   1:  PR[91,1] = PR[90,1] + -92.039;
   1:  PR[91,2] = PR[90,2] + -4.496;
   1:L PR[91] R[100]mm/sec CNT100;
   1:  PR[91,1] = PR[90,1] + -90.857;
   1:  PR[91,2] = PR[90,2] + -8.105;
   1:L PR[91] R[100]mm/sec CNT100;
   1:  PR[91,1] = PR[90,1] + -88.939;
   1:  PR[91,2] = PR[90,2] + -11.398;
   1:L PR[91] R[100]mm/sec CNT100TB   .50sec,CALL END_PUD;
   1:  PR[92] = PR[91];
   1:  PR[92,3] = PR[92,3] + 20;
   1:J PR[92] 10% FINE;
   1:  PR[91] = PR[90];
   1:  PR[91,1] = PR[90,1] + 75.472;
   1:  PR[91,2] = PR[90,2] + -19.127;
   1:  PR[91,3] = PR[90,3] + 22.295;
   1:  PR[92] = PR[91];
   1:  PR[92,3] = PR[92,3] + 20;
   1:J PR[92] 10% FINE;
   1:L PR[91] R[100]mm/sec CNT100;
   1:  CALL LASER_DRAHT_START;
   1:  PR[91,1] = PR[90,1] + 77.707;
   1:  PR[91,2] = PR[90,2] + -18.824;
   1:L PR[91] R[100]mm/sec CNT100;
   1:  PR[91,1] = PR[90,1] + 79.977;
   1:  PR[91,2] = PR[90,2] + -18.016;
   1:L PR[91] R[100]mm/sec CNT100;
   1:  PR[91,1] = PR[90,1] + 81.671;
   1:  PR[91,2] = PR[90,2] + -17.392;
   1:L PR[91] R[100]mm/sec CNT100;
   1:  PR[91,1] = PR[90,1] + 83.993;
   1:  PR[91,2] = PR[90,2] + -15.925;
   1:L PR[91] R[100]mm/sec CNT100;
   1:  PR[91,1] = PR[90,1] + 85.202;
   1:  PR[91,2] = PR[90,2] + -15.146;
   1:L PR[91] R[100]mm/sec CNT100;
   1:  PR[91,1] = PR[90,1] + 88.142;
   1:  PR[91,2] = PR[90,2] + -12.194;
   1:L PR[91] R[100]mm/sec CNT100;
   1:  PR[91,1] = PR[90,1] + 90.342;
   1:  PR[91,2] = PR[90,2] + -8.694;
   1:L PR[91] R[100]mm/sec CNT100;
   1:  PR[91,1] = PR[90,1] + 91.704;
   1:  PR[91,2] = PR[90,2] + -4.807;
   1:L PR[91] R[100]mm/sec CNT100;
   1:  PR[91,1] = PR[90,1] + 92.097;
   1:  PR[91,2] = PR[90,2] + -1.400;
   1:L PR[91] R[100]mm/sec CNT100;
   1:  PR[91,1] = PR[90,1] + 92.205;
   1:  PR[91,2] = PR[90,2] + -0.692;
   1:L PR[91] R[100]mm/sec CNT100;
   1:  PR[91,1] = PR[90,1] + 91.906;
   1:  PR[91,2] = PR[90,2] + 1.920;
   1:L PR[91] R[100]mm/sec CNT100;
   1:  PR[91,1] = PR[90,1] + 91.796;
   1:  PR[91,2] = PR[90,2] + 2.516;
   1:L PR[91] R[100]mm/sec CNT100;
   1:  PR[91,1] = PR[90,1] + 91.703;
   1:  PR[91,2] = PR[90,2] + 3.353;
   1:L PR[91] R[100]mm/sec CNT100;
   1:  PR[91,1] = PR[90,1] + 90.342;
   1:  PR[91,2] = PR[90,2] + 7.235;
   1:L PR[91] R[100]mm/sec CNT100;
   1:  PR[91,1] = PR[90,1] + 88.142;
   1:  PR[91,2] = PR[90,2] + 10.735;
   1:L PR[91] R[100]mm/sec CNT100;
   1:  PR[91,1] = PR[90,1] + 85.209;
   1:  PR[91,2] = PR[90,2] + 13.680;
   1:L PR[91] R[100]mm/sec CNT100;
   1:  PR[91,1] = PR[90,1] + 82.872;
   1:  PR[91,2] = PR[90,2] + 15.154;
   1:L PR[91] R[100]mm/sec CNT100;
   1:  PR[91,1] = PR[90,1] + 81.671;
   1:  PR[91,2] = PR[90,2] + 15.930;
   1:L PR[91] R[100]mm/sec CNT100;
   1:  PR[91,1] = PR[90,1] + 79.341;
   1:  PR[91,2] = PR[90,2] + 16.758;
   1:L PR[91] R[100]mm/sec CNT100;
   1:  PR[91,1] = PR[90,1] + 77.707;
   1:  PR[91,2] = PR[90,2] + 17.362;
   1:L PR[91] R[100]mm/sec CNT100;
   1:  PR[91,1] = PR[90,1] + 75.594;
   1:  PR[91,2] = PR[90,2] + 17.620;
   1:L PR[91] R[100]mm/sec CNT100;
   1:  PR[91,1] = PR[90,1] + 73.504;
   1:  PR[91,2] = PR[90,2] + 17.907;
   1:L PR[91] R[100]mm/sec CNT100;
   1:  PR[91,1] = PR[90,1] + 71.787;
   1:  PR[91,2] = PR[90,2] + 17.735;
   1:L PR[91] R[100]mm/sec CNT100;
   1:  PR[91,1] = PR[90,1] + 69.263;
   1:  PR[91,2] = PR[90,2] + 17.523;
   1:L PR[91] R[100]mm/sec CNT100;
   1:  PR[91,1] = PR[90,1] + 68.056;
   1:  PR[91,2] = PR[90,2] + 17.123;
   1:L PR[91] R[100]mm/sec CNT100;
   1:  PR[91,1] = PR[90,1] + 65.192;
   1:  PR[91,2] = PR[90,2] + 16.224;
   1:L PR[91] R[100]mm/sec CNT100;
   1:  PR[91,1] = PR[90,1] + 64.524;
   1:  PR[91,2] = PR[90,2] + 15.821;
   1:L PR[91] R[100]mm/sec CNT100;
   1:  PR[91,1] = PR[90,1] + 61.487;
   1:  PR[91,2] = PR[90,2] + 14.050;
   1:L PR[91] R[100]mm/sec CNT100;
   1:  PR[91,1] = PR[90,1] + 58.354;
   1:  PR[91,2] = PR[90,2] + 11.097;
   1:L PR[91] R[100]mm/sec CNT100;
   1:  PR[91,1] = PR[90,1] + 55.873;
   1:  PR[91,2] = PR[90,2] + 7.525;
   1:L PR[91] R[100]mm/sec CNT100;
   1:  PR[91,1] = PR[90,1] + 54.321;
   1:  PR[91,2] = PR[90,2] + 3.514;
   1:L PR[91] R[100]mm/sec CNT100;
   1:  PR[91,1] = PR[90,1] + 53.882;
   1:  PR[91,2] = PR[90,2] + 0.062;
   1:L PR[91] R[100]mm/sec CNT100;
   1:  PR[91,1] = PR[90,1] + 53.837;
   1:  PR[91,2] = PR[90,2] + -0.667;
   1:L PR[91] R[100]mm/sec CNT100;
   1:  PR[91,1] = PR[90,1] + 54.190;
   1:  PR[91,2] = PR[90,2] + -3.510;
   1:L PR[91] R[100]mm/sec CNT100;
   1:  PR[91,1] = PR[90,1] + 54.254;
   1:  PR[91,2] = PR[90,2] + -4.426;
   1:L PR[91] R[100]mm/sec CNT100;
   1:  PR[91,1] = PR[90,1] + 54.322;
   1:  PR[91,2] = PR[90,2] + -4.976;
   1:L PR[91] R[100]mm/sec CNT100;
   1:  PR[91,1] = PR[90,1] + 55.872;
   1:  PR[91,2] = PR[90,2] + -8.982;
   1:L PR[91] R[100]mm/sec CNT100;
   1:  PR[91,1] = PR[90,1] + 58.317;
   1:  PR[91,2] = PR[90,2] + -12.492;
   1:L PR[91] R[100]mm/sec CNT100;
   1:  PR[91,1] = PR[90,1] + 58.369;
   1:  PR[91,2] = PR[90,2] + -12.571;
   1:L PR[91] R[100]mm/sec CNT100;
   1:  PR[91,1] = PR[90,1] + 61.489;
   1:  PR[91,2] = PR[90,2] + -15.511;
   1:L PR[91] R[100]mm/sec CNT100;
   1:  PR[91,1] = PR[90,1] + 65.193;
   1:  PR[91,2] = PR[90,2] + -17.687;
   1:L PR[91] R[100]mm/sec CNT100;
   1:  PR[91,1] = PR[90,1] + 66.066;
   1:  PR[91,2] = PR[90,2] + -17.975;
   1:L PR[91] R[100]mm/sec CNT100;
   1:  PR[91,1] = PR[90,1] + 69.262;
   1:  PR[91,2] = PR[90,2] + -18.985;
   1:L PR[91] R[100]mm/sec CNT100;
   1:  PR[91,1] = PR[90,1] + 70.738;
   1:  PR[91,2] = PR[90,2] + -19.131;
   1:L PR[91] R[100]mm/sec CNT100;
   1:  PR[91,1] = PR[90,1] + 73.504;
   1:  PR[91,2] = PR[90,2] + -19.369;
   1:L PR[91] R[100]mm/sec CNT100;
   1:  PR[91,1] = PR[90,1] + 75.472;
   1:  PR[91,2] = PR[90,2] + -19.127;
   1:L PR[91] R[100]mm/sec CNT100TB   .50sec,CALL END_PUD;
   1:  PR[92] = PR[91];
   1:  PR[92,3] = PR[92,3] + 20;
   1:J PR[92] 10% FINE;
   1:  PR[91,1] = PR[90,1] + 37.828;
   1:  PR[91,2] = PR[90,2] + -13.861;
   1:  PR[92] = PR[91];
   1:  PR[92,3] = PR[92,3] + 20;
   1:J PR[92] 10% FINE;
   1:L PR[91] R[100]mm/sec CNT100;
   1:  CALL LASER_DRAHT_START;
   1:  PR[91,1] = PR[90,1] + 37.858;
   1:  PR[91,2] = PR[90,2] + -13.831;
   1:L PR[91] R[100]mm/sec CNT100;
   1:  PR[91,1] = PR[90,1] + 40.722;
   1:  PR[91,2] = PR[90,2] + -10.089;
   1:L PR[91] R[100]mm/sec CNT100;
   1:  PR[91,1] = PR[90,1] + 40.785;
   1:  PR[91,2] = PR[90,2] + -9.999;
   1:L PR[91] R[100]mm/sec CNT100;
   1:  PR[91,1] = PR[90,1] + 40.830;
   1:  PR[91,2] = PR[90,2] + -9.903;
   1:L PR[91] R[100]mm/sec CNT100;
   1:  PR[91,1] = PR[90,1] + 42.623;
   1:  PR[91,2] = PR[90,2] + -5.565;
   1:L PR[91] R[100]mm/sec CNT100;
   1:  PR[91,1] = PR[90,1] + 42.638;
   1:  PR[91,2] = PR[90,2] + -5.509;
   1:L PR[91] R[100]mm/sec CNT100;
   1:  PR[91,1] = PR[90,1] + 42.845;
   1:  PR[91,2] = PR[90,2] + -3.661;
   1:L PR[91] R[100]mm/sec CNT100;
   1:  PR[91,1] = PR[90,1] + 43.245;
   1:  PR[91,2] = PR[90,2] + -0.613;
   1:L PR[91] R[100]mm/sec CNT100;
   1:  PR[91,1] = PR[90,1] + 43.244;
   1:  PR[91,2] = PR[90,2] + -0.541;
   1:L PR[91] R[100]mm/sec CNT100;
   1:  PR[91,1] = PR[90,1] + 42.643;
   1:  PR[91,2] = PR[90,2] + 4.031;
   1:L PR[91] R[100]mm/sec CNT100;
   1:  PR[91,1] = PR[90,1] + 42.623;
   1:  PR[91,2] = PR[90,2] + 4.106;
   1:L PR[91] R[100]mm/sec CNT100;
   1:  PR[91,1] = PR[90,1] + 40.830;
   1:  PR[91,2] = PR[90,2] + 8.444;
   1:L PR[91] R[100]mm/sec CNT100;
   1:  PR[91,1] = PR[90,1] + 40.785;
   1:  PR[91,2] = PR[90,2] + 8.540;
   1:L PR[91] R[100]mm/sec CNT100;
   1:  PR[91,1] = PR[90,1] + 40.722;
   1:  PR[91,2] = PR[90,2] + 8.630;
   1:L PR[91] R[100]mm/sec CNT100;
   1:  PR[91,1] = PR[90,1] + 37.858;
   1:  PR[91,2] = PR[90,2] + 12.372;
   1:L PR[91] R[100]mm/sec CNT100;
   1:  PR[91,1] = PR[90,1] + 37.828;
   1:  PR[91,2] = PR[90,2] + 12.402;
   1:L PR[91] R[100]mm/sec CNT100;
   1:  PR[91,1] = PR[90,1] + 34.053;
   1:  PR[91,2] = PR[90,2] + 15.305;
   1:L PR[91] R[100]mm/sec CNT100;
   1:  PR[91,1] = PR[90,1] + 34.005;
   1:  PR[91,2] = PR[90,2] + 15.339;
   1:L PR[91] R[100]mm/sec CNT100;
   1:  PR[91,1] = PR[90,1] + 33.950;
   1:  PR[91,2] = PR[90,2] + 15.364;
   1:L PR[91] R[100]mm/sec CNT100;
   1:  PR[91,1] = PR[90,1] + 29.532;
   1:  PR[91,2] = PR[90,2] + 17.202;
   1:L PR[91] R[100]mm/sec CNT100;
   1:  PR[91,1] = PR[90,1] + 24.725;
   1:  PR[91,2] = PR[90,2] + 17.835;
   1:L PR[91] R[100]mm/sec CNT100;
   1:  PR[91,1] = PR[90,1] + 19.917;
   1:  PR[91,2] = PR[90,2] + 17.218;
   1:L PR[91] R[100]mm/sec CNT100;
   1:  PR[91,1] = PR[90,1] + 15.434;
   1:  PR[91,2] = PR[90,2] + 15.363;
   1:L PR[91] R[100]mm/sec CNT100;
   1:  PR[91,1] = PR[90,1] + 11.576;
   1:  PR[91,2] = PR[90,2] + 12.419;
   1:L PR[91] R[100]mm/sec CNT100;
   1:  PR[91,1] = PR[90,1] + 8.618;
   1:  PR[91,2] = PR[90,2] + 8.572;
   1:L PR[91] R[100]mm/sec CNT100;
   1:  PR[91,1] = PR[90,1] + 6.753;
   1:  PR[91,2] = PR[90,2] + 4.054;
   1:L PR[91] R[100]mm/sec CNT100;
   1:  PR[91,1] = PR[90,1] + 6.129;
   1:  PR[91,2] = PR[90,2] + -0.790;
   1:L PR[91] R[100]mm/sec CNT100;
   1:  PR[91,1] = PR[90,1] + 6.770;
   1:  PR[91,2] = PR[90,2] + -5.576;
   1:L PR[91] R[100]mm/sec CNT100;
   1:  PR[91,1] = PR[90,1] + 8.618;
   1:  PR[91,2] = PR[90,2] + -10.029;
   1:L PR[91] R[100]mm/sec CNT100;
   1:  PR[91,1] = PR[90,1] + 11.576;
   1:  PR[91,2] = PR[90,2] + -13.878;
   1:L PR[91] R[100]mm/sec CNT100;
   1:  PR[91,1] = PR[90,1] + 15.434;
   1:  PR[91,2] = PR[90,2] + -16.822;
   1:L PR[91] R[100]mm/sec CNT100;
   1:  PR[91,1] = PR[90,1] + 19.917;
   1:  PR[91,2] = PR[90,2] + -18.677;
   1:L PR[91] R[100]mm/sec CNT100;
   1:  PR[91,1] = PR[90,1] + 24.725;
   1:  PR[91,2] = PR[90,2] + -19.294;
   1:L PR[91] R[100]mm/sec CNT100;
   1:  PR[91,1] = PR[90,1] + 29.531;
   1:  PR[91,2] = PR[90,2] + -18.661;
   1:L PR[91] R[100]mm/sec CNT100;
   1:  PR[91,1] = PR[90,1] + 34.038;
   1:  PR[91,2] = PR[90,2] + -16.774;
   1:L PR[91] R[100]mm/sec CNT100;
   1:  PR[91,1] = PR[90,1] + 34.053;
   1:  PR[91,2] = PR[90,2] + -16.764;
   1:L PR[91] R[100]mm/sec CNT100;
   1:  PR[91,1] = PR[90,1] + 37.828;
   1:  PR[91,2] = PR[90,2] + -13.861;
   1:L PR[91] R[100]mm/sec CNT100TB   .50sec,CALL END_PUD;
   1:  PR[92] = PR[91];
   1:  PR[92,3] = PR[92,3] + 20;
   1:J PR[92] 10% FINE;
   1:  PR[91,1] = PR[90,1] + -5.907;
   1:  PR[91,2] = PR[90,2] + 3.403;
   1:  PR[92] = PR[91];
   1:  PR[92,3] = PR[92,3] + 20;
   1:J PR[92] 10% FINE;
   1:L PR[91] R[100]mm/sec CNT100;
   1:  CALL LASER_DRAHT_START;
   1:  PR[91,1] = PR[90,1] + -7.311;
   1:  PR[91,2] = PR[90,2] + 7.321;
   1:L PR[91] R[100]mm/sec CNT100;
   1:  PR[91,1] = PR[90,1] + -9.571;
   1:  PR[91,2] = PR[90,2] + 10.825;
   1:L PR[91] R[100]mm/sec CNT100;
   1:  PR[91,1] = PR[90,1] + -11.755;
   1:  PR[91,2] = PR[90,2] + 12.959;
   1:L PR[91] R[100]mm/sec CNT100;
   1:  PR[91,1] = PR[90,1] + -12.555;
   1:  PR[91,2] = PR[90,2] + 13.729;
   1:L PR[91] R[100]mm/sec CNT100;
   1:  PR[91,1] = PR[90,1] + -16.126;
   1:  PR[91,2] = PR[90,2] + 15.902;
   1:L PR[91] R[100]mm/sec CNT100;
   1:  PR[91,1] = PR[90,1] + -20.084;
   1:  PR[91,2] = PR[90,2] + 17.228;
   1:L PR[91] R[100]mm/sec CNT100;
   1:  PR[91,1] = PR[90,1] + -24.232;
   1:  PR[91,2] = PR[90,2] + 17.652;
   1:L PR[91] R[100]mm/sec CNT100;
   1:  PR[91,1] = PR[90,1] + -28.362;
   1:  PR[91,2] = PR[90,2] + 17.152;
   1:L PR[91] R[100]mm/sec CNT100;
   1:  PR[91,1] = PR[90,1] + -32.270;
   1:  PR[91,2] = PR[90,2] + 15.765;
   1:L PR[91] R[100]mm/sec CNT100;
   1:  PR[91,1] = PR[90,1] + -35.763;
   1:  PR[91,2] = PR[90,2] + 13.559;
   1:L PR[91] R[100]mm/sec CNT100;
   1:  PR[91,1] = PR[90,1] + -38.670;
   1:  PR[91,2] = PR[90,2] + 10.652;
   1:L PR[91] R[100]mm/sec CNT100;
   1:  PR[91,1] = PR[90,1] + -40.850;
   1:  PR[91,2] = PR[90,2] + 7.164;
   1:L PR[91] R[100]mm/sec CNT100;
   1:  PR[91,1] = PR[90,1] + -42.189;
   1:  PR[91,2] = PR[90,2] + 3.308;
   1:L PR[91] R[100]mm/sec CNT100;
   1:  PR[91,1] = PR[90,1] + -42.641;
   1:  PR[91,2] = PR[90,2] + -0.729;
   1:L PR[91] R[100]mm/sec CNT100;
   1:  PR[91,1] = PR[90,1] + -42.189;
   1:  PR[91,2] = PR[90,2] + -4.766;
   1:L PR[91] R[100]mm/sec CNT100;
   1:  PR[91,1] = PR[90,1] + -40.831;
   1:  PR[91,2] = PR[90,2] + -8.665;
   1:L PR[91] R[100]mm/sec CNT100;
   1:  PR[91,1] = PR[90,1] + -38.998;
   1:  PR[91,2] = PR[90,2] + -11.590;
   1:L PR[91] R[100]mm/sec CNT100;
   1:  PR[91,1] = PR[90,1] + -38.672;
   1:  PR[91,2] = PR[90,2] + -12.108;
   1:L PR[91] R[100]mm/sec CNT100;
   1:  PR[91,1] = PR[90,1] + -35.763;
   1:  PR[91,2] = PR[90,2] + -15.018;
   1:L PR[91] R[100]mm/sec CNT100;
   1:  PR[91,1] = PR[90,1] + -32.270;
   1:  PR[91,2] = PR[90,2] + -17.224;
   1:L PR[91] R[100]mm/sec CNT100;
   1:  PR[91,1] = PR[90,1] + -28.362;
   1:  PR[91,2] = PR[90,2] + -18.611;
   1:L PR[91] R[100]mm/sec CNT100;
   1:  PR[91,1] = PR[90,1] + -24.232;
   1:  PR[91,2] = PR[90,2] + -19.110;
   1:L PR[91] R[100]mm/sec CNT100;
   1:  PR[91,1] = PR[90,1] + -20.084;
   1:  PR[91,2] = PR[90,2] + -18.687;
   1:L PR[91] R[100]mm/sec CNT100;
   1:  PR[91,1] = PR[90,1] + -16.126;
   1:  PR[91,2] = PR[90,2] + -17.361;
   1:L PR[91] R[100]mm/sec CNT100;
   1:  PR[91,1] = PR[90,1] + -12.560;
   1:  PR[91,2] = PR[90,2] + -15.190;
   1:L PR[91] R[100]mm/sec CNT100;
   1:  PR[91,1] = PR[90,1] + -9.570;
   1:  PR[91,2] = PR[90,2] + -12.282;
   1:L PR[91] R[100]mm/sec CNT100;
   1:  PR[91,1] = PR[90,1] + -7.311;
   1:  PR[91,2] = PR[90,2] + -8.780;
   1:L PR[91] R[100]mm/sec CNT100;
   1:  PR[91,1] = PR[90,1] + -5.907;
   1:  PR[91,2] = PR[90,2] + -4.862;
   1:L PR[91] R[100]mm/sec CNT100;
   1:  PR[91,1] = PR[90,1] + -5.600;
   1:  PR[91,2] = PR[90,2] + -2.198;
   1:L PR[91] R[100]mm/sec CNT100;
   1:  PR[91,1] = PR[90,1] + -5.449;
   1:  PR[91,2] = PR[90,2] + -0.741;
   1:L PR[91] R[100]mm/sec CNT100;
   1:  PR[91,1] = PR[90,1] + -5.760;
   1:  PR[91,2] = PR[90,2] + 1.963;
   1:L PR[91] R[100]mm/sec CNT100;
   1:  PR[91,1] = PR[90,1] + -5.755;
   1:  PR[91,2] = PR[90,2] + 2.095;
   1:L PR[91] R[100]mm/sec CNT100;
   1:  PR[91,1] = PR[90,1] + -5.907;
   1:  PR[91,2] = PR[90,2] + 3.403;
   1:L PR[91] R[100]mm/sec CNT100TB   .50sec,CALL END_PUD;
   1:  PR[92] = PR[91];
   1:  PR[92,3] = PR[92,3] + 20;
   1:J PR[92] 10% FINE;
   1:  PR[91,1] = PR[90,1] + -73.284;
   1:  PR[91,2] = PR[90,2] + -18.980;
   1:  PR[92] = PR[91];
   1:  PR[92,3] = PR[92,3] + 20;
   1:J PR[92] 10% FINE;
   1:L PR[91] R[100]mm/sec CNT100;
   1:  CALL LASER_DRAHT_START;
   1:  PR[91,1] = PR[90,1] + -71.769;
   1:  PR[91,2] = PR[90,2] + -19.006;
   1:L PR[91] R[100]mm/sec CNT100;
   1:  PR[91,1] = PR[90,1] + -69.726;
   1:  PR[91,2] = PR[90,2] + -18.595;
   1:L PR[91] R[100]mm/sec CNT100;
   1:  PR[91,1] = PR[90,1] + -67.925;
   1:  PR[91,2] = PR[90,2] + -18.251;
   1:L PR[91] R[100]mm/sec CNT100;
   1:  PR[91,1] = PR[90,1] + -66.320;
   1:  PR[91,2] = PR[90,2] + -17.562;
   1:L PR[91] R[100]mm/sec CNT100;
   1:  PR[91,1] = PR[90,1] + -64.309;
   1:  PR[91,2] = PR[90,2] + -16.722;
   1:L PR[91] R[100]mm/sec CNT100;
   1:  PR[91,1] = PR[90,1] + -61.097;
   1:  PR[91,2] = PR[90,2] + -14.488;
   1:L PR[91] R[100]mm/sec CNT100;
   1:  PR[91,1] = PR[90,1] + -58.423;
   1:  PR[91,2] = PR[90,2] + -11.634;
   1:L PR[91] R[100]mm/sec CNT100;
   1:  PR[91,1] = PR[90,1] + -56.415;
   1:  PR[91,2] = PR[90,2] + -8.288;
   1:L PR[91] R[100]mm/sec CNT100;
   1:  PR[91,1] = PR[90,1] + -55.171;
   1:  PR[91,2] = PR[90,2] + -4.598;
   1:L PR[91] R[100]mm/sec CNT100;
   1:  PR[91,1] = PR[90,1] + -55.146;
   1:  PR[91,2] = PR[90,2] + -4.367;
   1:L PR[91] R[100]mm/sec CNT100;
   1:  PR[91,1] = PR[90,1] + -55.133;
   1:  PR[91,2] = PR[90,2] + -3.930;
   1:L PR[91] R[100]mm/sec CNT100;
   1:  PR[91,1] = PR[90,1] + -54.982;
   1:  PR[91,2] = PR[90,2] + -2.318;
   1:L PR[91] R[100]mm/sec CNT100;
   1:  PR[91,1] = PR[90,1] + -54.806;
   1:  PR[91,2] = PR[90,2] + -0.730;
   1:L PR[91] R[100]mm/sec CNT100;
   1:  PR[91,1] = PR[90,1] + -55.066;
   1:  PR[91,2] = PR[90,2] + 1.610;
   1:L PR[91] R[100]mm/sec CNT100;
   1:  PR[91,1] = PR[90,1] + -55.209;
   1:  PR[91,2] = PR[90,2] + 3.143;
   1:L PR[91] R[100]mm/sec CNT100;
   1:  PR[91,1] = PR[90,1] + -56.479;
   1:  PR[91,2] = PR[90,2] + 6.801;
   1:L PR[91] R[100]mm/sec CNT100;
   1:  PR[91,1] = PR[90,1] + -57.361;
   1:  PR[91,2] = PR[90,2] + 8.225;
   1:L PR[91] R[100]mm/sec CNT100;
   1:  PR[91,1] = PR[90,1] + -58.520;
   1:  PR[91,2] = PR[90,2] + 10.165;
   1:L PR[91] R[100]mm/sec CNT100;
   1:  PR[91,1] = PR[90,1] + -61.179;
   1:  PR[91,2] = PR[90,2] + 13.018;
   1:L PR[91] R[100]mm/sec CNT100;
   1:  PR[91,1] = PR[90,1] + -64.384;
   1:  PR[91,2] = PR[90,2] + 15.258;
   1:L PR[91] R[100]mm/sec CNT100;
   1:  PR[91,1] = PR[90,1] + -65.098;
   1:  PR[91,2] = PR[90,2] + 15.567;
   1:L PR[91] R[100]mm/sec CNT100;
   1:  PR[91,1] = PR[90,1] + -67.972;
   1:  PR[91,2] = PR[90,2] + 16.784;
   1:L PR[91] R[100]mm/sec CNT100;
   1:  PR[91,1] = PR[90,1] + -71.804;
   1:  PR[91,2] = PR[90,2] + 17.542;
   1:L PR[91] R[100]mm/sec CNT100;
   1:  PR[91,1] = PR[90,1] + -75.700;
   1:  PR[91,2] = PR[90,2] + 17.502;
   1:L PR[91] R[100]mm/sec CNT100;
   1:  PR[91,1] = PR[90,1] + -79.495;
   1:  PR[91,2] = PR[90,2] + 16.669;
   1:L PR[91] R[100]mm/sec CNT100;
   1:  PR[91,1] = PR[90,1] + -83.026;
   1:  PR[91,2] = PR[90,2] + 15.084;
   1:L PR[91] R[100]mm/sec CNT100;
   1:  PR[91,1] = PR[90,1] + -86.143;
   1:  PR[91,2] = PR[90,2] + 12.819;
   1:L PR[91] R[100]mm/sec CNT100;
   1:  PR[91,1] = PR[90,1] + -88.713;
   1:  PR[91,2] = PR[90,2] + 9.972;
   1:L PR[91] R[100]mm/sec CNT100;
   1:  PR[91,1] = PR[90,1] + -90.630;
   1:  PR[91,2] = PR[90,2] + 6.669;
   1:L PR[91] R[100]mm/sec CNT100;
   1:  PR[91,1] = PR[90,1] + -91.812;
   1:  PR[91,2] = PR[90,2] + 3.050;
   1:L PR[91] R[100]mm/sec CNT100;
   1:  PR[91,1] = PR[90,1] + -92.142;
   1:  PR[91,2] = PR[90,2] + -0.042;
   1:L PR[91] R[100]mm/sec CNT100;
   1:  PR[91,1] = PR[90,1] + -92.239;
   1:  PR[91,2] = PR[90,2] + -0.499;
   1:L PR[91] R[100]mm/sec CNT100;
   1:  PR[91,1] = PR[90,1] + -92.281;
   1:  PR[91,2] = PR[90,2] + -0.775;
   1:L PR[91] R[100]mm/sec CNT100;
   1:  PR[91,1] = PR[90,1] + -91.994;
   1:  PR[91,2] = PR[90,2] + -3.473;
   1:L PR[91] R[100]mm/sec CNT100;
   1:  PR[91,1] = PR[90,1] + -91.876;
   1:  PR[91,2] = PR[90,2] + -4.160;
   1:L PR[91] R[100]mm/sec CNT100;
   1:  PR[91,1] = PR[90,1] + -91.840;
   1:  PR[91,2] = PR[90,2] + -4.508;
   1:L PR[91] R[100]mm/sec CNT100;
   1:  PR[91,1] = PR[90,1] + -90.762;
   1:  PR[91,2] = PR[90,2] + -7.799;
   1:L PR[91] R[100]mm/sec CNT100;
   1:  PR[91,1] = PR[90,1] + -90.655;
   1:  PR[91,2] = PR[90,2] + -8.126;
   1:L PR[91] R[100]mm/sec CNT100;
   1:  PR[91,1] = PR[90,1] + -88.735;
   1:  PR[91,2] = PR[90,2] + -11.427;
   1:L PR[91] R[100]mm/sec CNT100;
   1:  PR[91,1] = PR[90,1] + -86.158;
   1:  PR[91,2] = PR[90,2] + -14.274;
   1:L PR[91] R[100]mm/sec CNT100;
   1:  PR[91,1] = PR[90,1] + -83.032;
   1:  PR[91,2] = PR[90,2] + -16.541;
   1:L PR[91] R[100]mm/sec CNT100;
   1:  PR[91,1] = PR[90,1] + -79.491;
   1:  PR[91,2] = PR[90,2] + -18.128;
   1:L PR[91] R[100]mm/sec CNT100;
   1:  PR[91,1] = PR[90,1] + -75.686;
   1:  PR[91,2] = PR[90,2] + -18.963;
   1:L PR[91] R[100]mm/sec CNT100;
   1:  PR[91,1] = PR[90,1] + -73.284;
   1:  PR[91,2] = PR[90,2] + -18.980;
   1:L PR[91] R[100]mm/sec CNT100TB   .50sec,CALL END_PUD;
   1:  PR[92] = PR[91];
   1:  PR[92,3] = PR[92,3] + 20;
   1:J PR[92] 10% FINE;
   1:  PR[91] = PR[90];
   1:  PR[91,1] = PR[90,1] + 73.272;
   1:  PR[91,2] = PR[90,2] + -19.473;
   1:  PR[91,3] = PR[90,3] + 23.595;
   1:  PR[92] = PR[91];
   1:  PR[92,3] = PR[92,3] + 20;
   1:J PR[92] 10% FINE;
   1:L PR[91] R[100]mm/sec CNT100;
   1:  CALL LASER_DRAHT_START;
   1:  PR[91,1] = PR[90,1] + 74.511;
   1:  PR[91,2] = PR[90,2] + -19.321;
   1:L PR[91] R[100]mm/sec CNT100;
   1:  PR[91,1] = PR[90,1] + 77.495;
   1:  PR[91,2] = PR[90,2] + -18.917;
   1:L PR[91] R[100]mm/sec CNT100;
   1:  PR[91,1] = PR[90,1] + 79.122;
   1:  PR[91,2] = PR[90,2] + -18.338;
   1:L PR[91] R[100]mm/sec CNT100;
   1:  PR[91,1] = PR[90,1] + 81.475;
   1:  PR[91,2] = PR[90,2] + -17.471;
   1:L PR[91] R[100]mm/sec CNT100;
   1:  PR[91,1] = PR[90,1] + 83.259;
   1:  PR[91,2] = PR[90,2] + -16.344;
   1:L PR[91] R[100]mm/sec CNT100;
   1:  PR[91,1] = PR[90,1] + 85.018;
   1:  PR[91,2] = PR[90,2] + -15.210;
   1:L PR[91] R[100]mm/sec CNT100;
   1:  PR[91,1] = PR[90,1] + 87.967;
   1:  PR[91,2] = PR[90,2] + -12.243;
   1:L PR[91] R[100]mm/sec CNT100;
   1:  PR[91,1] = PR[90,1] + 90.174;
   1:  PR[91,2] = PR[90,2] + -8.726;
   1:L PR[91] R[100]mm/sec CNT100;
   1:  PR[91,1] = PR[90,1] + 91.540;
   1:  PR[91,2] = PR[90,2] + -4.823;
   1:L PR[91] R[100]mm/sec CNT100;
   1:  PR[91,1] = PR[90,1] + 91.871;
   1:  PR[91,2] = PR[90,2] + -1.951;
   1:L PR[91] R[100]mm/sec CNT100;
   1:  PR[91,1] = PR[90,1] + 92.063;
   1:  PR[91,2] = PR[90,2] + -0.692;
   1:L PR[91] R[100]mm/sec CNT100;
   1:  PR[91,1] = PR[90,1] + 91.859;
   1:  PR[91,2] = PR[90,2] + 1.092;
   1:L PR[91] R[100]mm/sec CNT100;
   1:  PR[91,1] = PR[90,1] + 91.690;
   1:  PR[91,2] = PR[90,2] + 2.004;
   1:L PR[91] R[100]mm/sec CNT100;
   1:  PR[91,1] = PR[90,1] + 91.538;
   1:  PR[91,2] = PR[90,2] + 3.369;
   1:L PR[91] R[100]mm/sec CNT100;
   1:  PR[91,1] = PR[90,1] + 90.174;
   1:  PR[91,2] = PR[90,2] + 7.267;
   1:L PR[91] R[100]mm/sec CNT100;
   1:  PR[91,1] = PR[90,1] + 87.967;
   1:  PR[91,2] = PR[90,2] + 10.784;
   1:L PR[91] R[100]mm/sec CNT100;
   1:  PR[91,1] = PR[90,1] + 85.025;
   1:  PR[91,2] = PR[90,2] + 13.744;
   1:L PR[91] R[100]mm/sec CNT100;
   1:  PR[91,1] = PR[90,1] + 83.157;
   1:  PR[91,2] = PR[90,2] + 14.922;
   1:L PR[91] R[100]mm/sec CNT100;
   1:  PR[91,1] = PR[90,1] + 81.475;
   1:  PR[91,2] = PR[90,2] + 16.009;
   1:L PR[91] R[100]mm/sec CNT100;
   1:  PR[91,1] = PR[90,1] + 79.690;
   1:  PR[91,2] = PR[90,2] + 16.643;
   1:L PR[91] R[100]mm/sec CNT100;
   1:  PR[91,1] = PR[90,1] + 77.495;
   1:  PR[91,2] = PR[90,2] + 17.456;
   1:L PR[91] R[100]mm/sec CNT100;
   1:  PR[91,1] = PR[90,1] + 75.986;
   1:  PR[91,2] = PR[90,2] + 17.640;
   1:L PR[91] R[100]mm/sec CNT100;
   1:  PR[91,1] = PR[90,1] + 73.270;
   1:  PR[91,2] = PR[90,2] + 18.012;
   1:L PR[91] R[100]mm/sec CNT100;
   1:  PR[91,1] = PR[90,1] + 72.197;
   1:  PR[91,2] = PR[90,2] + 17.905;
   1:L PR[91] R[100]mm/sec CNT100;
   1:  PR[91,1] = PR[90,1] + 69.002;
   1:  PR[91,2] = PR[90,2] + 17.636;
   1:L PR[91] R[100]mm/sec CNT100;
   1:  PR[91,1] = PR[90,1] + 68.451;
   1:  PR[91,2] = PR[90,2] + 17.453;
   1:L PR[91] R[100]mm/sec CNT100;
   1:  PR[91,1] = PR[90,1] + 64.888;
   1:  PR[91,2] = PR[90,2] + 16.335;
   1:L PR[91] R[100]mm/sec CNT100;
   1:  PR[91,1] = PR[90,1] + 63.034;
   1:  PR[91,2] = PR[90,2] + 15.250;
   1:L PR[91] R[100]mm/sec CNT100;
   1:  PR[91,1] = PR[90,1] + 61.049;
   1:  PR[91,2] = PR[90,2] + 14.153;
   1:L PR[91] R[100]mm/sec CNT100;
   1:  PR[91,1] = PR[90,1] + 58.225;
   1:  PR[91,2] = PR[90,2] + 11.615;
   1:L PR[91] R[100]mm/sec CNT100;
   1:  PR[91,1] = PR[90,1] + 57.749;
   1:  PR[91,2] = PR[90,2] + 11.204;
   1:L PR[91] R[100]mm/sec CNT100;
   1:  PR[91,1] = PR[90,1] + 55.897;
   1:  PR[91,2] = PR[90,2] + 8.536;
   1:L PR[91] R[100]mm/sec CNT100;
   1:  PR[91,1] = PR[90,1] + 55.238;
   1:  PR[91,2] = PR[90,2] + 7.619;
   1:L PR[91] R[100]mm/sec CNT100;
   1:  PR[91,1] = PR[90,1] + 54.224;
   1:  PR[91,2] = PR[90,2] + 4.984;
   1:L PR[91] R[100]mm/sec CNT100;
   1:  PR[91,1] = PR[90,1] + 53.660;
   1:  PR[91,2] = PR[90,2] + 3.563;
   1:L PR[91] R[100]mm/sec CNT100;
   1:  PR[91,1] = PR[90,1] + 53.352;
   1:  PR[91,2] = PR[90,2] + 1.137;
   1:L PR[91] R[100]mm/sec CNT100;
   1:  PR[91,1] = PR[90,1] + 53.240;
   1:  PR[91,2] = PR[90,2] + -0.667;
   1:L PR[91] R[100]mm/sec CNT100;
   1:  PR[91,1] = PR[90,1] + 53.292;
   1:  PR[91,2] = PR[90,2] + -1.083;
   1:L PR[91] R[100]mm/sec CNT100;
   1:  PR[91,1] = PR[90,1] + 53.446;
   1:  PR[91,2] = PR[90,2] + -3.288;
   1:L PR[91] R[100]mm/sec CNT100;
   1:  PR[91,1] = PR[90,1] + 53.662;
   1:  PR[91,2] = PR[90,2] + -5.031;
   1:L PR[91] R[100]mm/sec CNT100;
   1:  PR[91,1] = PR[90,1] + 55.241;
   1:  PR[91,2] = PR[90,2] + -9.088;
   1:L PR[91] R[100]mm/sec CNT100;
   1:  PR[91,1] = PR[90,1] + 57.194;
   1:  PR[91,2] = PR[90,2] + -11.892;
   1:L PR[91] R[100]mm/sec CNT100;
   1:  PR[91,1] = PR[90,1] + 57.748;
   1:  PR[91,2] = PR[90,2] + -12.667;
   1:L PR[91] R[100]mm/sec CNT100;
   1:  PR[91,1] = PR[90,1] + 61.046;
   1:  PR[91,2] = PR[90,2] + -15.610;
   1:L PR[91] R[100]mm/sec CNT100;
   1:  PR[91,1] = PR[90,1] + 63.034;
   1:  PR[91,2] = PR[90,2] + -16.709;
   1:L PR[91] R[100]mm/sec CNT100;
   1:  PR[91,1] = PR[90,1] + 64.891;
   1:  PR[91,2] = PR[90,2] + -17.795;
   1:L PR[91] R[100]mm/sec CNT100;
   1:  PR[91,1] = PR[90,1] + 68.993;
   1:  PR[91,2] = PR[90,2] + -19.095;
   1:L PR[91] R[100]mm/sec CNT100;
   1:  PR[91,1] = PR[90,1] + 73.272;
   1:  PR[91,2] = PR[90,2] + -19.473;
   1:L PR[91] R[100]mm/sec CNT100TB   .50sec,CALL END_PUD;
   1:  PR[92] = PR[91];
   1:  PR[92,3] = PR[92,3] + 20;
   1:J PR[92] 10% FINE;
   1:  PR[91,1] = PR[90,1] + 34.001;
   1:  PR[91,2] = PR[90,2] + 15.387;
   1:  PR[92] = PR[91];
   1:  PR[92,3] = PR[92,3] + 20;
   1:J PR[92] 10% FINE;
   1:L PR[91] R[100]mm/sec CNT100;
   1:  CALL LASER_DRAHT_START;
   1:  PR[91,1] = PR[90,1] + 29.511;
   1:  PR[91,2] = PR[90,2] + 17.264;
   1:L PR[91] R[100]mm/sec CNT100;
   1:  PR[91,1] = PR[90,1] + 24.682;
   1:  PR[91,2] = PR[90,2] + 17.919;
   1:L PR[91] R[100]mm/sec CNT100;
   1:  PR[91,1] = PR[90,1] + 19.849;
   1:  PR[91,2] = PR[90,2] + 17.301;
   1:L PR[91] R[100]mm/sec CNT100;
   1:  PR[91,1] = PR[90,1] + 15.329;
   1:  PR[91,2] = PR[90,2] + 15.450;
   1:L PR[91] R[100]mm/sec CNT100;
   1:  PR[91,1] = PR[90,1] + 11.444;
   1:  PR[91,2] = PR[90,2] + 12.492;
   1:L PR[91] R[100]mm/sec CNT100;
   1:  PR[91,1] = PR[90,1] + 8.460;
   1:  PR[91,2] = PR[90,2] + 8.624;
   1:L PR[91] R[100]mm/sec CNT100;
   1:  PR[91,1] = PR[90,1] + 6.582;
   1:  PR[91,2] = PR[90,2] + 4.114;
   1:L PR[91] R[100]mm/sec CNT100;
   1:  PR[91,1] = PR[90,1] + 5.940;
   1:  PR[91,2] = PR[90,2] + -0.729;
   1:L PR[91] R[100]mm/sec CNT100;
   1:  PR[91,1] = PR[90,1] + 6.582;
   1:  PR[91,2] = PR[90,2] + -5.573;
   1:L PR[91] R[100]mm/sec CNT100;
   1:  PR[91,1] = PR[90,1] + 8.460;
   1:  PR[91,2] = PR[90,2] + -10.084;
   1:L PR[91] R[100]mm/sec CNT100;
   1:  PR[91,1] = PR[90,1] + 11.445;
   1:  PR[91,2] = PR[90,2] + -13.951;
   1:L PR[91] R[100]mm/sec CNT100;
   1:  PR[91,1] = PR[90,1] + 15.330;
   1:  PR[91,2] = PR[90,2] + -16.909;
   1:L PR[91] R[100]mm/sec CNT100;
   1:  PR[91,1] = PR[90,1] + 19.846;
   1:  PR[91,2] = PR[90,2] + -18.759;
   1:L PR[91] R[100]mm/sec CNT100;
   1:  PR[91,1] = PR[90,1] + 24.683;
   1:  PR[91,2] = PR[90,2] + -19.377;
   1:L PR[91] R[100]mm/sec CNT100;
   1:  PR[91,1] = PR[90,1] + 29.511;
   1:  PR[91,2] = PR[90,2] + -18.723;
   1:L PR[91] R[100]mm/sec CNT100;
   1:  PR[91,1] = PR[90,1] + 34.002;
   1:  PR[91,2] = PR[90,2] + -16.846;
   1:L PR[91] R[100]mm/sec CNT100;
   1:  PR[91,1] = PR[90,1] + 37.853;
   1:  PR[91,2] = PR[90,2] + -13.877;
   1:L PR[91] R[100]mm/sec CNT100;
   1:  PR[91,1] = PR[90,1] + 40.801;
   1:  PR[91,2] = PR[90,2] + -10.023;
   1:L PR[91] R[100]mm/sec CNT100;
   1:  PR[91,1] = PR[90,1] + 42.658;
   1:  PR[91,2] = PR[90,2] + -5.521;
   1:L PR[91] R[100]mm/sec CNT100;
   1:  PR[91,1] = PR[90,1] + 43.285;
   1:  PR[91,2] = PR[90,2] + -0.729;
   1:L PR[91] R[100]mm/sec CNT100;
   1:  PR[91,1] = PR[90,1] + 42.659;
   1:  PR[91,2] = PR[90,2] + 4.062;
   1:L PR[91] R[100]mm/sec CNT100;
   1:  PR[91,1] = PR[90,1] + 40.787;
   1:  PR[91,2] = PR[90,2] + 8.584;
   1:L PR[91] R[100]mm/sec CNT100;
   1:  PR[91,1] = PR[90,1] + 37.851;
   1:  PR[91,2] = PR[90,2] + 12.419;
   1:L PR[91] R[100]mm/sec CNT100;
   1:  PR[91,1] = PR[90,1] + 34.001;
   1:  PR[91,2] = PR[90,2] + 15.387;
   1:L PR[91] R[100]mm/sec CNT100TB   .50sec,CALL END_PUD;
   1:  PR[92] = PR[91];
   1:  PR[92,3] = PR[92,3] + 20;
   1:J PR[92] 10% FINE;
   1:  PR[91,1] = PR[90,1] + -17.097;
   1:  PR[91,2] = PR[90,2] + -17.840;
   1:  PR[92] = PR[91];
   1:  PR[92,3] = PR[92,3] + 20;
   1:J PR[92] 10% FINE;
   1:L PR[91] R[100]mm/sec CNT100;
   1:  CALL LASER_DRAHT_START;
   1:  PR[91,1] = PR[90,1] + -15.887;
   1:  PR[91,2] = PR[90,2] + -17.446;
   1:L PR[91] R[100]mm/sec CNT100;
   1:  PR[91,1] = PR[90,1] + -13.580;
   1:  PR[91,2] = PR[90,2] + -16.033;
   1:L PR[91] R[100]mm/sec CNT100;
   1:  PR[91,1] = PR[90,1] + -12.297;
   1:  PR[91,2] = PR[90,2] + -15.265;
   1:L PR[91] R[100]mm/sec CNT100;
   1:  PR[91,1] = PR[90,1] + -9.292;
   1:  PR[91,2] = PR[90,2] + -12.348;
   1:L PR[91] R[100]mm/sec CNT100;
   1:  PR[91,1] = PR[90,1] + -7.017;
   1:  PR[91,2] = PR[90,2] + -8.827;
   1:L PR[91] R[100]mm/sec CNT100;
   1:  PR[91,1] = PR[90,1] + -5.603;
   1:  PR[91,2] = PR[90,2] + -4.887;
   1:L PR[91] R[100]mm/sec CNT100;
   1:  PR[91,1] = PR[90,1] + -5.363;
   1:  PR[91,2] = PR[90,2] + -2.813;
   1:L PR[91] R[100]mm/sec CNT100;
   1:  PR[91,1] = PR[90,1] + -5.148;
   1:  PR[91,2] = PR[90,2] + -0.741;
   1:L PR[91] R[100]mm/sec CNT100;
   1:  PR[91,1] = PR[90,1] + -5.385;
   1:  PR[91,2] = PR[90,2] + 1.312;
   1:L PR[91] R[100]mm/sec CNT100;
   1:  PR[91,1] = PR[90,1] + -5.378;
   1:  PR[91,2] = PR[90,2] + 1.494;
   1:L PR[91] R[100]mm/sec CNT100;
   1:  PR[91,1] = PR[90,1] + -5.603;
   1:  PR[91,2] = PR[90,2] + 3.428;
   1:L PR[91] R[100]mm/sec CNT100;
   1:  PR[91,1] = PR[90,1] + -7.018;
   1:  PR[91,2] = PR[90,2] + 7.371;
   1:L PR[91] R[100]mm/sec CNT100;
   1:  PR[91,1] = PR[90,1] + -8.249;
   1:  PR[91,2] = PR[90,2] + 9.288;
   1:L PR[91] R[100]mm/sec CNT100;
   1:  PR[91,1] = PR[90,1] + -9.289;
   1:  PR[91,2] = PR[90,2] + 10.887;
   1:L PR[91] R[100]mm/sec CNT100;
   1:  PR[91,1] = PR[90,1] + -12.302;
   1:  PR[91,2] = PR[90,2] + 13.811;
   1:L PR[91] R[100]mm/sec CNT100;
   1:  PR[91,1] = PR[90,1] + -15.890;
   1:  PR[91,2] = PR[90,2] + 15.989;
   1:L PR[91] R[100]mm/sec CNT100;
   1:  PR[91,1] = PR[90,1] + -19.870;
   1:  PR[91,2] = PR[90,2] + 17.317;
   1:L PR[91] R[100]mm/sec CNT100;
   1:  PR[91,1] = PR[90,1] + -24.038;
   1:  PR[91,2] = PR[90,2] + 17.738;
   1:L PR[91] R[100]mm/sec CNT100;
   1:  PR[91,1] = PR[90,1] + -28.187;
   1:  PR[91,2] = PR[90,2] + 17.232;
   1:L PR[91] R[100]mm/sec CNT100;
   1:  PR[91,1] = PR[90,1] + -32.112;
   1:  PR[91,2] = PR[90,2] + 15.834;
   1:L PR[91] R[100]mm/sec CNT100;
   1:  PR[91,1] = PR[90,1] + -35.275;
   1:  PR[91,2] = PR[90,2] + 13.838;
   1:L PR[91] R[100]mm/sec CNT100;
   1:  PR[91,1] = PR[90,1] + -35.612;
   1:  PR[91,2] = PR[90,2] + 13.622;
   1:L PR[91] R[100]mm/sec CNT100;
   1:  PR[91,1] = PR[90,1] + -38.535;
   1:  PR[91,2] = PR[90,2] + 10.694;
   1:L PR[91] R[100]mm/sec CNT100;
   1:  PR[91,1] = PR[90,1] + -40.725;
   1:  PR[91,2] = PR[90,2] + 7.211;
   1:L PR[91] R[100]mm/sec CNT100;
   1:  PR[91,1] = PR[90,1] + -42.082;
   1:  PR[91,2] = PR[90,2] + 3.340;
   1:L PR[91] R[100]mm/sec CNT100;
   1:  PR[91,1] = PR[90,1] + -42.545;
   1:  PR[91,2] = PR[90,2] + -0.746;
   1:L PR[91] R[100]mm/sec CNT100;
   1:  PR[91,1] = PR[90,1] + -42.560;
   1:  PR[91,2] = PR[90,2] + -0.819;
   1:L PR[91] R[100]mm/sec CNT100;
   1:  PR[91,1] = PR[90,1] + -42.412;
   1:  PR[91,2] = PR[90,2] + -2.127;
   1:L PR[91] R[100]mm/sec CNT100;
   1:  PR[91,1] = PR[90,1] + -42.093;
   1:  PR[91,2] = PR[90,2] + -4.697;
   1:L PR[91] R[100]mm/sec CNT100;
   1:  PR[91,1] = PR[90,1] + -42.081;
   1:  PR[91,2] = PR[90,2] + -4.800;
   1:L PR[91] R[100]mm/sec CNT100;
   1:  PR[91,1] = PR[90,1] + -40.725;
   1:  PR[91,2] = PR[90,2] + -8.670;
   1:L PR[91] R[100]mm/sec CNT100;
   1:  PR[91,1] = PR[90,1] + -38.535;
   1:  PR[91,2] = PR[90,2] + -12.153;
   1:L PR[91] R[100]mm/sec CNT100;
   1:  PR[91,1] = PR[90,1] + -35.617;
   1:  PR[91,2] = PR[90,2] + -15.076;
   1:L PR[91] R[100]mm/sec CNT100;
   1:  PR[91,1] = PR[90,1] + -32.111;
   1:  PR[91,2] = PR[90,2] + -17.294;
   1:L PR[91] R[100]mm/sec CNT100;
   1:  PR[91,1] = PR[90,1] + -28.187;
   1:  PR[91,2] = PR[90,2] + -18.691;
   1:L PR[91] R[100]mm/sec CNT100;
   1:  PR[91,1] = PR[90,1] + -24.041;
   1:  PR[91,2] = PR[90,2] + -19.196;
   1:L PR[91] R[100]mm/sec CNT100;
   1:  PR[91,1] = PR[90,1] + -20.916;
   1:  PR[91,2] = PR[90,2] + -18.872;
   1:L PR[91] R[100]mm/sec CNT100;
   1:  PR[91,1] = PR[90,1] + -19.865;
   1:  PR[91,2] = PR[90,2] + -18.774;
   1:L PR[91] R[100]mm/sec CNT100;
   1:  PR[91,1] = PR[90,1] + -17.097;
   1:  PR[91,2] = PR[90,2] + -17.840;
   1:L PR[91] R[100]mm/sec CNT100TB   .50sec,CALL END_PUD;
   1:  PR[92] = PR[91];
   1:  PR[92,3] = PR[92,3] + 20;
   1:J PR[92] 10% FINE;
   1:  PR[91,1] = PR[90,1] + -54.561;
   1:  PR[91,2] = PR[90,2] + 2.063;
   1:  PR[92] = PR[91];
   1:  PR[92,3] = PR[92,3] + 20;
   1:J PR[92] 10% FINE;
   1:L PR[91] R[100]mm/sec CNT100;
   1:  CALL LASER_DRAHT_START;
   1:  PR[91,1] = PR[90,1] + -54.685;
   1:  PR[91,2] = PR[90,2] + 3.153;
   1:L PR[91] R[100]mm/sec CNT100;
   1:  PR[91,1] = PR[90,1] + -55.975;
   1:  PR[91,2] = PR[90,2] + 6.856;
   1:L PR[91] R[100]mm/sec CNT100;
   1:  PR[91,1] = PR[90,1] + -58.056;
   1:  PR[91,2] = PR[90,2] + 10.208;
   1:L PR[91] R[100]mm/sec CNT100;
   1:  PR[91,1] = PR[90,1] + -60.821;
   1:  PR[91,2] = PR[90,2] + 13.062;
   1:L PR[91] R[100]mm/sec CNT100;
   1:  PR[91,1] = PR[90,1] + -62.566;
   1:  PR[91,2] = PR[90,2] + 14.231;
   1:L PR[91] R[100]mm/sec CNT100;
   1:  PR[91,1] = PR[90,1] + -64.123;
   1:  PR[91,2] = PR[90,2] + 15.317;
   1:L PR[91] R[100]mm/sec CNT100;
   1:  PR[91,1] = PR[90,1] + -67.733;
   1:  PR[91,2] = PR[90,2] + 16.848;
   1:L PR[91] R[100]mm/sec CNT100;
   1:  PR[91,1] = PR[90,1] + -71.582;
   1:  PR[91,2] = PR[90,2] + 17.604;
   1:L PR[91] R[100]mm/sec CNT100;
   1:  PR[91,1] = PR[90,1] + -72.515;
   1:  PR[91,2] = PR[90,2] + 17.599;
   1:L PR[91] R[100]mm/sec CNT100;
   1:  PR[91,1] = PR[90,1] + -75.485;
   1:  PR[91,2] = PR[90,2] + 17.559;
   1:L PR[91] R[100]mm/sec CNT100;
   1:  PR[91,1] = PR[90,1] + -79.292;
   1:  PR[91,2] = PR[90,2] + 16.720;
   1:L PR[91] R[100]mm/sec CNT100;
   1:  PR[91,1] = PR[90,1] + -82.832;
   1:  PR[91,2] = PR[90,2] + 15.127;
   1:L PR[91] R[100]mm/sec CNT100;
   1:  PR[91,1] = PR[90,1] + -85.955;
   1:  PR[91,2] = PR[90,2] + 12.854;
   1:L PR[91] R[100]mm/sec CNT100;
   1:  PR[91,1] = PR[90,1] + -88.530;
   1:  PR[91,2] = PR[90,2] + 9.999;
   1:L PR[91] R[100]mm/sec CNT100;
   1:  PR[91,1] = PR[90,1] + -90.450;
   1:  PR[91,2] = PR[90,2] + 6.687;
   1:L PR[91] R[100]mm/sec CNT100;
   1:  PR[91,1] = PR[90,1] + -91.634;
   1:  PR[91,2] = PR[90,2] + 3.058;
   1:L PR[91] R[100]mm/sec CNT100;
   1:  PR[91,1] = PR[90,1] + -91.911;
   1:  PR[91,2] = PR[90,2] + 0.465;
   1:L PR[91] R[100]mm/sec CNT100;
   1:  PR[91,1] = PR[90,1] + -91.994;
   1:  PR[91,2] = PR[90,2] + 0.072;
   1:L PR[91] R[100]mm/sec CNT100;
   1:  PR[91,1] = PR[90,1] + -92.123;
   1:  PR[91,2] = PR[90,2] + -0.775;
   1:L PR[91] R[100]mm/sec CNT100;
   1:  PR[91,1] = PR[90,1] + -91.948;
   1:  PR[91,2] = PR[90,2] + -2.426;
   1:L PR[91] R[100]mm/sec CNT100;
   1:  PR[91,1] = PR[90,1] + -91.797;
   1:  PR[91,2] = PR[90,2] + -3.381;
   1:L PR[91] R[100]mm/sec CNT100;
   1:  PR[91,1] = PR[90,1] + -91.731;
   1:  PR[91,2] = PR[90,2] + -3.660;
   1:L PR[91] R[100]mm/sec CNT100;
   1:  PR[91,1] = PR[90,1] + -91.642;
   1:  PR[91,2] = PR[90,2] + -4.517;
   1:L PR[91] R[100]mm/sec CNT100;
   1:  PR[91,1] = PR[90,1] + -90.701;
   1:  PR[91,2] = PR[90,2] + -7.387;
   1:L PR[91] R[100]mm/sec CNT100;
   1:  PR[91,1] = PR[90,1] + -90.455;
   1:  PR[91,2] = PR[90,2] + -8.145;
   1:L PR[91] R[100]mm/sec CNT100;
   1:  PR[91,1] = PR[90,1] + -88.530;
   1:  PR[91,2] = PR[90,2] + -11.455;
   1:L PR[91] R[100]mm/sec CNT100;
   1:  PR[91,1] = PR[90,1] + -85.949;
   1:  PR[91,2] = PR[90,2] + -14.312;
   1:L PR[91] R[100]mm/sec CNT100;
   1:  PR[91,1] = PR[90,1] + -82.816;
   1:  PR[91,2] = PR[90,2] + -16.588;
   1:L PR[91] R[100]mm/sec CNT100;
   1:  PR[91,1] = PR[90,1] + -79.264;
   1:  PR[91,2] = PR[90,2] + -18.184;
   1:L PR[91] R[100]mm/sec CNT100;
   1:  PR[91,1] = PR[90,1] + -75.449;
   1:  PR[91,2] = PR[90,2] + -19.025;
   1:L PR[91] R[100]mm/sec CNT100;
   1:  PR[91,1] = PR[90,1] + -73.578;
   1:  PR[91,2] = PR[90,2] + -19.039;
   1:L PR[91] R[100]mm/sec CNT100;
   1:  PR[91,1] = PR[90,1] + -71.520;
   1:  PR[91,2] = PR[90,2] + -19.074;
   1:L PR[91] R[100]mm/sec CNT100;
   1:  PR[91,1] = PR[90,1] + -70.024;
   1:  PR[91,2] = PR[90,2] + -18.773;
   1:L PR[91] R[100]mm/sec CNT100;
   1:  PR[91,1] = PR[90,1] + -67.652;
   1:  PR[91,2] = PR[90,2] + -18.321;
   1:L PR[91] R[100]mm/sec CNT100;
   1:  PR[91,1] = PR[90,1] + -64.027;
   1:  PR[91,2] = PR[90,2] + -16.794;
   1:L PR[91] R[100]mm/sec CNT100;
   1:  PR[91,1] = PR[90,1] + -60.793;
   1:  PR[91,2] = PR[90,2] + -14.551;
   1:L PR[91] R[100]mm/sec CNT100;
   1:  PR[91,1] = PR[90,1] + -58.102;
   1:  PR[91,2] = PR[90,2] + -11.685;
   1:L PR[91] R[100]mm/sec CNT100;
   1:  PR[91,1] = PR[90,1] + -56.062;
   1:  PR[91,2] = PR[90,2] + -8.314;
   1:L PR[91] R[100]mm/sec CNT100;
   1:  PR[91,1] = PR[90,1] + -54.754;
   1:  PR[91,2] = PR[90,2] + -4.602;
   1:L PR[91] R[100]mm/sec CNT100;
   1:  PR[91,1] = PR[90,1] + -54.327;
   1:  PR[91,2] = PR[90,2] + -0.916;
   1:L PR[91] R[100]mm/sec CNT100;
   1:  PR[91,1] = PR[90,1] + -54.315;
   1:  PR[91,2] = PR[90,2] + -0.745;
   1:L PR[91] R[100]mm/sec CNT100;
   1:  PR[91,1] = PR[90,1] + -54.561;
   1:  PR[91,2] = PR[90,2] + 2.063;
   1:L PR[91] R[100]mm/sec CNT100TB   .50sec,CALL END_PUD;
   1:  PR[92] = PR[91];
   1:  PR[92,3] = PR[92,3] + 20;
   1:J PR[92] 10% FINE;
   1:  PR[91] = PR[90];
   1:  PR[91,1] = PR[90,1] + 53.000;
   1:  PR[91,2] = PR[90,2] + 3.621;
   1:  PR[91,3] = PR[90,3] + 24.895;
   1:  PR[92] = PR[91];
   1:  PR[92,3] = PR[92,3] + 20;
   1:J PR[92] 10% FINE;
   1:L PR[91] R[100]mm/sec CNT100;
   1:  CALL LASER_DRAHT_START;
   1:  PR[91,1] = PR[90,1] + 52.821;
   1:  PR[91,2] = PR[90,2] + 2.212;
   1:L PR[91] R[100]mm/sec CNT100;
   1:  PR[91,1] = PR[90,1] + 52.724;
   1:  PR[91,2] = PR[90,2] + 0.636;
   1:L PR[91] R[100]mm/sec CNT100;
   1:  PR[91,1] = PR[90,1] + 52.542;
   1:  PR[91,2] = PR[90,2] + -0.787;
   1:L PR[91] R[100]mm/sec CNT100;
   1:  PR[91,1] = PR[90,1] + 52.637;
   1:  PR[91,2] = PR[90,2] + -2.151;
   1:L PR[91] R[100]mm/sec CNT100;
   1:  PR[91,1] = PR[90,1] + 53.002;
   1:  PR[91,2] = PR[90,2] + -5.092;
   1:L PR[91] R[100]mm/sec CNT100;
   1:  PR[91,1] = PR[90,1] + 53.615;
   1:  PR[91,2] = PR[90,2] + -6.680;
   1:L PR[91] R[100]mm/sec CNT100;
   1:  PR[91,1] = PR[90,1] + 54.608;
   1:  PR[91,2] = PR[90,2] + -9.191;
   1:L PR[91] R[100]mm/sec CNT100;
   1:  PR[91,1] = PR[90,1] + 55.896;
   1:  PR[91,2] = PR[90,2] + -11.041;
   1:L PR[91] R[100]mm/sec CNT100;
   1:  PR[91,1] = PR[90,1] + 57.163;
   1:  PR[91,2] = PR[90,2] + -12.813;
   1:L PR[91] R[100]mm/sec CNT100;
   1:  PR[91,1] = PR[90,1] + 59.431;
   1:  PR[91,2] = PR[90,2] + -14.842;
   1:L PR[91] R[100]mm/sec CNT100;
   1:  PR[91,1] = PR[90,1] + 60.497;
   1:  PR[91,2] = PR[90,2] + -15.768;
   1:L PR[91] R[100]mm/sec CNT100;
   1:  PR[91,1] = PR[90,1] + 64.431;
   1:  PR[91,2] = PR[90,2] + -17.929;
   1:L PR[91] R[100]mm/sec CNT100;
   1:  PR[91,1] = PR[90,1] + 68.003;
   1:  PR[91,2] = PR[90,2] + -18.978;
   1:L PR[91] R[100]mm/sec CNT100;
   1:  PR[91,1] = PR[90,1] + 68.730;
   1:  PR[91,2] = PR[90,2] + -19.208;
   1:L PR[91] R[100]mm/sec CNT100;
   1:  PR[91,1] = PR[90,1] + 73.036;
   1:  PR[91,2] = PR[90,2] + -19.579;
   1:L PR[91] R[100]mm/sec CNT100;
   1:  PR[91,1] = PR[90,1] + 73.551;
   1:  PR[91,2] = PR[90,2] + -19.516;
   1:L PR[91] R[100]mm/sec CNT100;
   1:  PR[91,1] = PR[90,1] + 77.283;
   1:  PR[91,2] = PR[90,2] + -19.011;
   1:L PR[91] R[100]mm/sec CNT100;
   1:  PR[91,1] = PR[90,1] + 78.268;
   1:  PR[91,2] = PR[90,2] + -18.660;
   1:L PR[91] R[100]mm/sec CNT100;
   1:  PR[91,1] = PR[90,1] + 81.280;
   1:  PR[91,2] = PR[90,2] + -17.550;
   1:L PR[91] R[100]mm/sec CNT100;
   1:  PR[91,1] = PR[90,1] + 82.526;
   1:  PR[91,2] = PR[90,2] + -16.763;
   1:L PR[91] R[100]mm/sec CNT100;
   1:  PR[91,1] = PR[90,1] + 84.834;
   1:  PR[91,2] = PR[90,2] + -15.274;
   1:L PR[91] R[100]mm/sec CNT100;
   1:  PR[91,1] = PR[90,1] + 87.792;
   1:  PR[91,2] = PR[90,2] + -12.292;
   1:L PR[91] R[100]mm/sec CNT100;
   1:  PR[91,1] = PR[90,1] + 90.007;
   1:  PR[91,2] = PR[90,2] + -8.757;
   1:L PR[91] R[100]mm/sec CNT100;
   1:  PR[91,1] = PR[90,1] + 90.734;
   1:  PR[91,2] = PR[90,2] + -6.688;
   1:L PR[91] R[100]mm/sec CNT100;
   1:  PR[91,1] = PR[90,1] + 91.375;
   1:  PR[91,2] = PR[90,2] + -4.842;
   1:L PR[91] R[100]mm/sec CNT100;
   1:  PR[91,1] = PR[90,1] + 91.645;
   1:  PR[91,2] = PR[90,2] + -2.502;
   1:L PR[91] R[100]mm/sec CNT100;
   1:  PR[91,1] = PR[90,1] + 91.921;
   1:  PR[91,2] = PR[90,2] + -0.692;
   1:L PR[91] R[100]mm/sec CNT100;
   1:  PR[91,1] = PR[90,1] + 91.811;
   1:  PR[91,2] = PR[90,2] + 0.265;
   1:L PR[91] R[100]mm/sec CNT100;
   1:  PR[91,1] = PR[90,1] + 91.584;
   1:  PR[91,2] = PR[90,2] + 1.492;
   1:L PR[91] R[100]mm/sec CNT100;
   1:  PR[91,1] = PR[90,1] + 91.374;
   1:  PR[91,2] = PR[90,2] + 3.385;
   1:L PR[91] R[100]mm/sec CNT100;
   1:  PR[91,1] = PR[90,1] + 90.006;
   1:  PR[91,2] = PR[90,2] + 7.300;
   1:L PR[91] R[100]mm/sec CNT100;
   1:  PR[91,1] = PR[90,1] + 87.795;
   1:  PR[91,2] = PR[90,2] + 10.829;
   1:L PR[91] R[100]mm/sec CNT100;
   1:  PR[91,1] = PR[90,1] + 86.441;
   1:  PR[91,2] = PR[90,2] + 12.181;
   1:L PR[91] R[100]mm/sec CNT100;
   1:  PR[91,1] = PR[90,1] + 84.838;
   1:  PR[91,2] = PR[90,2] + 13.810;
   1:L PR[91] R[100]mm/sec CNT100;
   1:  PR[91,1] = PR[90,1] + 83.443;
   1:  PR[91,2] = PR[90,2] + 14.690;
   1:L PR[91] R[100]mm/sec CNT100;
   1:  PR[91,1] = PR[90,1] + 81.280;
   1:  PR[91,2] = PR[90,2] + 16.088;
   1:L PR[91] R[100]mm/sec CNT100;
   1:  PR[91,1] = PR[90,1] + 80.040;
   1:  PR[91,2] = PR[90,2] + 16.529;
   1:L PR[91] R[100]mm/sec CNT100;
   1:  PR[91,1] = PR[90,1] + 77.283;
   1:  PR[91,2] = PR[90,2] + 17.549;
   1:L PR[91] R[100]mm/sec CNT100;
   1:  PR[91,1] = PR[90,1] + 76.379;
   1:  PR[91,2] = PR[90,2] + 17.659;
   1:L PR[91] R[100]mm/sec CNT100;
   1:  PR[91,1] = PR[90,1] + 73.023;
   1:  PR[91,2] = PR[90,2] + 18.119;
   1:L PR[91] R[100]mm/sec CNT100;
   1:  PR[91,1] = PR[90,1] + 68.730;
   1:  PR[91,2] = PR[90,2] + 17.749;
   1:L PR[91] R[100]mm/sec CNT100;
   1:  PR[91,1] = PR[90,1] + 68.004;
   1:  PR[91,2] = PR[90,2] + 17.519;
   1:L PR[91] R[100]mm/sec CNT100;
   1:  PR[91,1] = PR[90,1] + 64.435;
   1:  PR[91,2] = PR[90,2] + 16.472;
   1:L PR[91] R[100]mm/sec CNT100;
   1:  PR[91,1] = PR[90,1] + 61.289;
   1:  PR[91,2] = PR[90,2] + 14.723;
   1:L PR[91] R[100]mm/sec CNT100;
   1:  PR[91,1] = PR[90,1] + 60.499;
   1:  PR[91,2] = PR[90,2] + 14.306;
   1:L PR[91] R[100]mm/sec CNT100;
   1:  PR[91,1] = PR[90,1] + 58.310;
   1:  PR[91,2] = PR[90,2] + 12.338;
   1:L PR[91] R[100]mm/sec CNT100;
   1:  PR[91,1] = PR[90,1] + 57.164;
   1:  PR[91,2] = PR[90,2] + 11.349;
   1:L PR[91] R[100]mm/sec CNT100;
   1:  PR[91,1] = PR[90,1] + 55.827;
   1:  PR[91,2] = PR[90,2] + 9.423;
   1:L PR[91] R[100]mm/sec CNT100;
   1:  PR[91,1] = PR[90,1] + 54.608;
   1:  PR[91,2] = PR[90,2] + 7.726;
   1:L PR[91] R[100]mm/sec CNT100;
   1:  PR[91,1] = PR[90,1] + 53.945;
   1:  PR[91,2] = PR[90,2] + 6.004;
   1:L PR[91] R[100]mm/sec CNT100;
   1:  PR[91,1] = PR[90,1] + 53.000;
   1:  PR[91,2] = PR[90,2] + 3.621;
   1:L PR[91] R[100]mm/sec CNT100TB   .50sec,CALL END_PUD;
   1:  PR[92] = PR[91];
   1:  PR[92,3] = PR[92,3] + 20;
   1:J PR[92] 10% FINE;
   1:  PR[91,1] = PR[90,1] + 8.268;
   1:  PR[91,2] = PR[90,2] + 8.694;
   1:  PR[92] = PR[91];
   1:  PR[92,3] = PR[92,3] + 20;
   1:J PR[92] 10% FINE;
   1:L PR[91] R[100]mm/sec CNT100;
   1:  CALL LASER_DRAHT_START;
   1:  PR[91,1] = PR[90,1] + 6.376;
   1:  PR[91,2] = PR[90,2] + 4.150;
   1:L PR[91] R[100]mm/sec CNT100;
   1:  PR[91,1] = PR[90,1] + 5.730;
   1:  PR[91,2] = PR[90,2] + -0.729;
   1:L PR[91] R[100]mm/sec CNT100;
   1:  PR[91,1] = PR[90,1] + 6.377;
   1:  PR[91,2] = PR[90,2] + -5.610;
   1:L PR[91] R[100]mm/sec CNT100;
   1:  PR[91,1] = PR[90,1] + 8.269;
   1:  PR[91,2] = PR[90,2] + -10.154;
   1:L PR[91] R[100]mm/sec CNT100;
   1:  PR[91,1] = PR[90,1] + 11.275;
   1:  PR[91,2] = PR[90,2] + -14.051;
   1:L PR[91] R[100]mm/sec CNT100;
   1:  PR[91,1] = PR[90,1] + 15.188;
   1:  PR[91,2] = PR[90,2] + -17.031;
   1:L PR[91] R[100]mm/sec CNT100;
   1:  PR[91,1] = PR[90,1] + 19.740;
   1:  PR[91,2] = PR[90,2] + -18.897;
   1:L PR[91] R[100]mm/sec CNT100;
   1:  PR[91,1] = PR[90,1] + 20.215;
   1:  PR[91,2] = PR[90,2] + -18.959;
   1:L PR[91] R[100]mm/sec CNT100;
   1:  PR[91,1] = PR[90,1] + 24.608;
   1:  PR[91,2] = PR[90,2] + -19.520;
   1:L PR[91] R[100]mm/sec CNT100;
   1:  PR[91,1] = PR[90,1] + 29.471;
   1:  PR[91,2] = PR[90,2] + -18.863;
   1:L PR[91] R[100]mm/sec CNT100;
   1:  PR[91,1] = PR[90,1] + 34.002;
   1:  PR[91,2] = PR[90,2] + -16.973;
   1:L PR[91] R[100]mm/sec CNT100;
   1:  PR[91,1] = PR[90,1] + 34.223;
   1:  PR[91,2] = PR[90,2] + -16.805;
   1:L PR[91] R[100]mm/sec CNT100;
   1:  PR[91,1] = PR[90,1] + 37.872;
   1:  PR[91,2] = PR[90,2] + -13.991;
   1:L PR[91] R[100]mm/sec CNT100;
   1:  PR[91,1] = PR[90,1] + 40.847;
   1:  PR[91,2] = PR[90,2] + -10.106;
   1:L PR[91] R[100]mm/sec CNT100;
   1:  PR[91,1] = PR[90,1] + 42.712;
   1:  PR[91,2] = PR[90,2] + -5.626;
   1:L PR[91] R[100]mm/sec CNT100;
   1:  PR[91,1] = PR[90,1] + 42.747;
   1:  PR[91,2] = PR[90,2] + -5.491;
   1:L PR[91] R[100]mm/sec CNT100;
   1:  PR[91,1] = PR[90,1] + 43.338;
   1:  PR[91,2] = PR[90,2] + -0.994;
   1:L PR[91] R[100]mm/sec CNT100;
   1:  PR[91,1] = PR[90,1] + 43.358;
   1:  PR[91,2] = PR[90,2] + -0.772;
   1:L PR[91] R[100]mm/sec CNT100;
   1:  PR[91,1] = PR[90,1] + 42.777;
   1:  PR[91,2] = PR[90,2] + 3.645;
   1:L PR[91] R[100]mm/sec CNT100;
   1:  PR[91,1] = PR[90,1] + 42.740;
   1:  PR[91,2] = PR[90,2] + 4.053;
   1:L PR[91] R[100]mm/sec CNT100;
   1:  PR[91,1] = PR[90,1] + 42.704;
   1:  PR[91,2] = PR[90,2] + 4.191;
   1:L PR[91] R[100]mm/sec CNT100;
   1:  PR[91,1] = PR[90,1] + 40.933;
   1:  PR[91,2] = PR[90,2] + 8.481;
   1:L PR[91] R[100]mm/sec CNT100;
   1:  PR[91,1] = PR[90,1] + 40.872;
   1:  PR[91,2] = PR[90,2] + 8.614;
   1:L PR[91] R[100]mm/sec CNT100;
   1:  PR[91,1] = PR[90,1] + 37.870;
   1:  PR[91,2] = PR[90,2] + 12.534;
   1:L PR[91] R[100]mm/sec CNT100;
   1:  PR[91,1] = PR[90,1] + 33.990;
   1:  PR[91,2] = PR[90,2] + 15.520;
   1:L PR[91] R[100]mm/sec CNT100;
   1:  PR[91,1] = PR[90,1] + 29.789;
   1:  PR[91,2] = PR[90,2] + 17.276;
   1:L PR[91] R[100]mm/sec CNT100;
   1:  PR[91,1] = PR[90,1] + 29.476;
   1:  PR[91,2] = PR[90,2] + 17.404;
   1:L PR[91] R[100]mm/sec CNT100;
   1:  PR[91,1] = PR[90,1] + 24.605;
   1:  PR[91,2] = PR[90,2] + 18.061;
   1:L PR[91] R[100]mm/sec CNT100;
   1:  PR[91,1] = PR[90,1] + 19.733;
   1:  PR[91,2] = PR[90,2] + 17.436;
   1:L PR[91] R[100]mm/sec CNT100;
   1:  PR[91,1] = PR[90,1] + 15.692;
   1:  PR[91,2] = PR[90,2] + 15.781;
   1:L PR[91] R[100]mm/sec CNT100;
   1:  PR[91,1] = PR[90,1] + 15.188;
   1:  PR[91,2] = PR[90,2] + 15.573;
   1:L PR[91] R[100]mm/sec CNT100;
   1:  PR[91,1] = PR[90,1] + 11.273;
   1:  PR[91,2] = PR[90,2] + 12.590;
   1:L PR[91] R[100]mm/sec CNT100;
   1:  PR[91,1] = PR[90,1] + 8.268;
   1:  PR[91,2] = PR[90,2] + 8.694;
   1:L PR[91] R[100]mm/sec CNT100TB   .50sec,CALL END_PUD;
   1:  PR[92] = PR[91];
   1:  PR[92,3] = PR[92,3] + 20;
   1:J PR[92] 10% FINE;
   1:  PR[91,1] = PR[90,1] + -28.012;
   1:  PR[91,2] = PR[90,2] + 17.312;
   1:  PR[92] = PR[91];
   1:  PR[92,3] = PR[92,3] + 20;
   1:J PR[92] 10% FINE;
   1:L PR[91] R[100]mm/sec CNT100;
   1:  CALL LASER_DRAHT_START;
   1:  PR[91,1] = PR[90,1] + -31.954;
   1:  PR[91,2] = PR[90,2] + 15.904;
   1:L PR[91] R[100]mm/sec CNT100;
   1:  PR[91,1] = PR[90,1] + -34.716;
   1:  PR[91,2] = PR[90,2] + 14.161;
   1:L PR[91] R[100]mm/sec CNT100;
   1:  PR[91,1] = PR[90,1] + -35.466;
   1:  PR[91,2] = PR[90,2] + 13.679;
   1:L PR[91] R[100]mm/sec CNT100;
   1:  PR[91,1] = PR[90,1] + -38.398;
   1:  PR[91,2] = PR[90,2] + 10.738;
   1:L PR[91] R[100]mm/sec CNT100;
   1:  PR[91,1] = PR[90,1] + -40.595;
   1:  PR[91,2] = PR[90,2] + 7.241;
   1:L PR[91] R[100]mm/sec CNT100;
   1:  PR[91,1] = PR[90,1] + -41.956;
   1:  PR[91,2] = PR[90,2] + 3.355;
   1:L PR[91] R[100]mm/sec CNT100;
   1:  PR[91,1] = PR[90,1] + -42.372;
   1:  PR[91,2] = PR[90,2] + -0.312;
   1:L PR[91] R[100]mm/sec CNT100;
   1:  PR[91,1] = PR[90,1] + -42.457;
   1:  PR[91,2] = PR[90,2] + -0.729;
   1:L PR[91] R[100]mm/sec CNT100;
   1:  PR[91,1] = PR[90,1] + -42.014;
   1:  PR[91,2] = PR[90,2] + -4.284;
   1:L PR[91] R[100]mm/sec CNT100;
   1:  PR[91,1] = PR[90,1] + -41.955;
   1:  PR[91,2] = PR[90,2] + -4.815;
   1:L PR[91] R[100]mm/sec CNT100;
   1:  PR[91,1] = PR[90,1] + -40.595;
   1:  PR[91,2] = PR[90,2] + -8.700;
   1:L PR[91] R[100]mm/sec CNT100;
   1:  PR[91,1] = PR[90,1] + -38.398;
   1:  PR[91,2] = PR[90,2] + -12.197;
   1:L PR[91] R[100]mm/sec CNT100;
   1:  PR[91,1] = PR[90,1] + -35.470;
   1:  PR[91,2] = PR[90,2] + -15.134;
   1:L PR[91] R[100]mm/sec CNT100;
   1:  PR[91,1] = PR[90,1] + -31.952;
   1:  PR[91,2] = PR[90,2] + -17.363;
   1:L PR[91] R[100]mm/sec CNT100;
   1:  PR[91,1] = PR[90,1] + -28.016;
   1:  PR[91,2] = PR[90,2] + -18.769;
   1:L PR[91] R[100]mm/sec CNT100;
   1:  PR[91,1] = PR[90,1] + -25.155;
   1:  PR[91,2] = PR[90,2] + -19.111;
   1:L PR[91] R[100]mm/sec CNT100;
   1:  PR[91,1] = PR[90,1] + -23.842;
   1:  PR[91,2] = PR[90,2] + -19.282;
   1:L PR[91] R[100]mm/sec CNT100;
   1:  PR[91,1] = PR[90,1] + -21.201;
   1:  PR[91,2] = PR[90,2] + -19.008;
   1:L PR[91] R[100]mm/sec CNT100;
   1:  PR[91,1] = PR[90,1] + -19.654;
   1:  PR[91,2] = PR[90,2] + -18.864;
   1:L PR[91] R[100]mm/sec CNT100;
   1:  PR[91,1] = PR[90,1] + -17.358;
   1:  PR[91,2] = PR[90,2] + -18.089;
   1:L PR[91] R[100]mm/sec CNT100;
   1:  PR[91,1] = PR[90,1] + -15.653;
   1:  PR[91,2] = PR[90,2] + -17.534;
   1:L PR[91] R[100]mm/sec CNT100;
   1:  PR[91,1] = PR[90,1] + -13.789;
   1:  PR[91,2] = PR[90,2] + -16.393;
   1:L PR[91] R[100]mm/sec CNT100;
   1:  PR[91,1] = PR[90,1] + -12.044;
   1:  PR[91,2] = PR[90,2] + -15.348;
   1:L PR[91] R[100]mm/sec CNT100;
   1:  PR[91,1] = PR[90,1] + -10.644;
   1:  PR[91,2] = PR[90,2] + -13.979;
   1:L PR[91] R[100]mm/sec CNT100;
   1:  PR[91,1] = PR[90,1] + -9.012;
   1:  PR[91,2] = PR[90,2] + -12.411;
   1:L PR[91] R[100]mm/sec CNT100;
   1:  PR[91,1] = PR[90,1] + -6.723;
   1:  PR[91,2] = PR[90,2] + -8.875;
   1:L PR[91] R[100]mm/sec CNT100;
   1:  PR[91,1] = PR[90,1] + -5.298;
   1:  PR[91,2] = PR[90,2] + -4.912;
   1:L PR[91] R[100]mm/sec CNT100;
   1:  PR[91,1] = PR[90,1] + -5.127;
   1:  PR[91,2] = PR[90,2] + -3.428;
   1:L PR[91] R[100]mm/sec CNT100;
   1:  PR[91,1] = PR[90,1] + -4.848;
   1:  PR[91,2] = PR[90,2] + -0.741;
   1:L PR[91] R[100]mm/sec CNT100;
   1:  PR[91,1] = PR[90,1] + -5.010;
   1:  PR[91,2] = PR[90,2] + 0.662;
   1:L PR[91] R[100]mm/sec CNT100;
   1:  PR[91,1] = PR[90,1] + -5.001;
   1:  PR[91,2] = PR[90,2] + 0.893;
   1:L PR[91] R[100]mm/sec CNT100;
   1:  PR[91,1] = PR[90,1] + -5.298;
   1:  PR[91,2] = PR[90,2] + 3.453;
   1:L PR[91] R[100]mm/sec CNT100;
   1:  PR[91,1] = PR[90,1] + -6.723;
   1:  PR[91,2] = PR[90,2] + 7.416;
   1:L PR[91] R[100]mm/sec CNT100;
   1:  PR[91,1] = PR[90,1] + -9.014;
   1:  PR[91,2] = PR[90,2] + 10.955;
   1:L PR[91] R[100]mm/sec CNT100;
   1:  PR[91,1] = PR[90,1] + -12.047;
   1:  PR[91,2] = PR[90,2] + 13.894;
   1:L PR[91] R[100]mm/sec CNT100;
   1:  PR[91,1] = PR[90,1] + -13.845;
   1:  PR[91,2] = PR[90,2] + 14.994;
   1:L PR[91] R[100]mm/sec CNT100;
   1:  PR[91,1] = PR[90,1] + -15.653;
   1:  PR[91,2] = PR[90,2] + 16.077;
   1:L PR[91] R[100]mm/sec CNT100;
   1:  PR[91,1] = PR[90,1] + -17.900;
   1:  PR[91,2] = PR[90,2] + 16.835;
   1:L PR[91] R[100]mm/sec CNT100;
   1:  PR[91,1] = PR[90,1] + -19.654;
   1:  PR[91,2] = PR[90,2] + 17.407;
   1:L PR[91] R[100]mm/sec CNT100;
   1:  PR[91,1] = PR[90,1] + -22.274;
   1:  PR[91,2] = PR[90,2] + 17.678;
   1:L PR[91] R[100]mm/sec CNT100;
   1:  PR[91,1] = PR[90,1] + -23.839;
   1:  PR[91,2] = PR[90,2] + 17.825;
   1:L PR[91] R[100]mm/sec CNT100;
   1:  PR[91,1] = PR[90,1] + -28.012;
   1:  PR[91,2] = PR[90,2] + 17.312;
   1:L PR[91] R[100]mm/sec CNT100TB   .50sec,CALL END_PUD;
   1:  PR[92] = PR[91];
   1:  PR[92,3] = PR[92,3] + 20;
   1:J PR[92] 10% FINE;
   1:  PR[91,1] = PR[90,1] + -91.965;
   1:  PR[91,2] = PR[90,2] + -0.775;
   1:  PR[92] = PR[91];
   1:  PR[92,3] = PR[92,3] + 20;
   1:J PR[92] 10% FINE;
   1:L PR[91] R[100]mm/sec CNT100;
   1:  CALL LASER_DRAHT_START;
   1:  PR[91,1] = PR[90,1] + -91.902;
   1:  PR[91,2] = PR[90,2] + -1.365;
   1:L PR[91] R[100]mm/sec CNT100;
   1:  PR[91,1] = PR[90,1] + -91.671;
   1:  PR[91,2] = PR[90,2] + -2.832;
   1:L PR[91] R[100]mm/sec CNT100;
   1:  PR[91,1] = PR[90,1] + -91.580;
   1:  PR[91,2] = PR[90,2] + -3.221;
   1:L PR[91] R[100]mm/sec CNT100;
   1:  PR[91,1] = PR[90,1] + -91.443;
   1:  PR[91,2] = PR[90,2] + -4.526;
   1:L PR[91] R[100]mm/sec CNT100;
   1:  PR[91,1] = PR[90,1] + -90.641;
   1:  PR[91,2] = PR[90,2] + -6.975;
   1:L PR[91] R[100]mm/sec CNT100;
   1:  PR[91,1] = PR[90,1] + -90.254;
   1:  PR[91,2] = PR[90,2] + -8.164;
   1:L PR[91] R[100]mm/sec CNT100;
   1:  PR[91,1] = PR[90,1] + -88.326;
   1:  PR[91,2] = PR[90,2] + -11.484;
   1:L PR[91] R[100]mm/sec CNT100;
   1:  PR[91,1] = PR[90,1] + -85.739;
   1:  PR[91,2] = PR[90,2] + -14.350;
   1:L PR[91] R[100]mm/sec CNT100;
   1:  PR[91,1] = PR[90,1] + -82.599;
   1:  PR[91,2] = PR[90,2] + -16.635;
   1:L PR[91] R[100]mm/sec CNT100;
   1:  PR[91,1] = PR[90,1] + -79.038;
   1:  PR[91,2] = PR[90,2] + -18.239;
   1:L PR[91] R[100]mm/sec CNT100;
   1:  PR[91,1] = PR[90,1] + -75.212;
   1:  PR[91,2] = PR[90,2] + -19.088;
   1:L PR[91] R[100]mm/sec CNT100;
   1:  PR[91,1] = PR[90,1] + -73.873;
   1:  PR[91,2] = PR[90,2] + -19.097;
   1:L PR[91] R[100]mm/sec CNT100;
   1:  PR[91,1] = PR[90,1] + -71.262;
   1:  PR[91,2] = PR[90,2] + -19.142;
   1:L PR[91] R[100]mm/sec CNT100;
   1:  PR[91,1] = PR[90,1] + -67.387;
   1:  PR[91,2] = PR[90,2] + -18.392;
   1:L PR[91] R[100]mm/sec CNT100;
   1:  PR[91,1] = PR[90,1] + -63.742;
   1:  PR[91,2] = PR[90,2] + -16.862;
   1:L PR[91] R[100]mm/sec CNT100;
   1:  PR[91,1] = PR[90,1] + -60.834;
   1:  PR[91,2] = PR[90,2] + -14.852;
   1:L PR[91] R[100]mm/sec CNT100;
   1:  PR[91,1] = PR[90,1] + -60.435;
   1:  PR[91,2] = PR[90,2] + -14.589;
   1:L PR[91] R[100]mm/sec CNT100;
   1:  PR[91,1] = PR[90,1] + -57.617;
   1:  PR[91,2] = PR[90,2] + -11.727;
   1:L PR[91] R[100]mm/sec CNT100;
   1:  PR[91,1] = PR[90,1] + -55.494;
   1:  PR[91,2] = PR[90,2] + -8.359;
   1:L PR[91] R[100]mm/sec CNT100;
   1:  PR[91,1] = PR[90,1] + -54.176;
   1:  PR[91,2] = PR[90,2] + -4.634;
   1:L PR[91] R[100]mm/sec CNT100;
   1:  PR[91,1] = PR[90,1] + -53.844;
   1:  PR[91,2] = PR[90,2] + -1.761;
   1:L PR[91] R[100]mm/sec CNT100;
   1:  PR[91,1] = PR[90,1] + -53.770;
   1:  PR[91,2] = PR[90,2] + -0.745;
   1:L PR[91] R[100]mm/sec CNT100;
   1:  PR[91,1] = PR[90,1] + -53.934;
   1:  PR[91,2] = PR[90,2] + 1.126;
   1:L PR[91] R[100]mm/sec CNT100;
   1:  PR[91,1] = PR[90,1] + -54.167;
   1:  PR[91,2] = PR[90,2] + 3.182;
   1:L PR[91] R[100]mm/sec CNT100;
   1:  PR[91,1] = PR[90,1] + -55.471;
   1:  PR[91,2] = PR[90,2] + 6.911;
   1:L PR[91] R[100]mm/sec CNT100;
   1:  PR[91,1] = PR[90,1] + -57.572;
   1:  PR[91,2] = PR[90,2] + 10.284;
   1:L PR[91] R[100]mm/sec CNT100;
   1:  PR[91,1] = PR[90,1] + -60.362;
   1:  PR[91,2] = PR[90,2] + 13.153;
   1:L PR[91] R[100]mm/sec CNT100;
   1:  PR[91,1] = PR[90,1] + -63.710;
   1:  PR[91,2] = PR[90,2] + 15.390;
   1:L PR[91] R[100]mm/sec CNT100;
   1:  PR[91,1] = PR[90,1] + -67.467;
   1:  PR[91,2] = PR[90,2] + 16.910;
   1:L PR[91] R[100]mm/sec CNT100;
   1:  PR[91,1] = PR[90,1] + -71.350;
   1:  PR[91,2] = PR[90,2] + 17.665;
   1:L PR[91] R[100]mm/sec CNT100;
   1:  PR[91,1] = PR[90,1] + -75.273;
   1:  PR[91,2] = PR[90,2] + 17.615;
   1:L PR[91] R[100]mm/sec CNT100;
   1:  PR[91,1] = PR[90,1] + -79.090;
   1:  PR[91,2] = PR[90,2] + 16.770;
   1:L PR[91] R[100]mm/sec CNT100;
   1:  PR[91,1] = PR[90,1] + -82.637;
   1:  PR[91,2] = PR[90,2] + 15.170;
   1:L PR[91] R[100]mm/sec CNT100;
   1:  PR[91,1] = PR[90,1] + -85.767;
   1:  PR[91,2] = PR[90,2] + 12.888;
   1:L PR[91] R[100]mm/sec CNT100;
   1:  PR[91,1] = PR[90,1] + -88.347;
   1:  PR[91,2] = PR[90,2] + 10.025;
   1:L PR[91] R[100]mm/sec CNT100;
   1:  PR[91,1] = PR[90,1] + -90.271;
   1:  PR[91,2] = PR[90,2] + 6.704;
   1:L PR[91] R[100]mm/sec CNT100;
   1:  PR[91,1] = PR[90,1] + -91.456;
   1:  PR[91,2] = PR[90,2] + 3.067;
   1:L PR[91] R[100]mm/sec CNT100;
   1:  PR[91,1] = PR[90,1] + -91.680;
   1:  PR[91,2] = PR[90,2] + 0.971;
   1:L PR[91] R[100]mm/sec CNT100;
   1:  PR[91,1] = PR[90,1] + -91.750;
   1:  PR[91,2] = PR[90,2] + 0.643;
   1:L PR[91] R[100]mm/sec CNT100;
   1:  PR[91,1] = PR[90,1] + -91.965;
   1:  PR[91,2] = PR[90,2] + -0.775;
   1:L PR[91] R[100]mm/sec CNT100TB   .50sec,CALL END_PUD;
   1:  PR[92] = PR[91];
   1:  PR[92,3] = PR[92,3] + 20;
   1:J PR[92] 10% FINE;
   1:  PR[91] = PR[90];
   1:  PR[91,1] = PR[90,1] + 58.395;
   1:  PR[91,2] = PR[90,2] + 13.062;
   1:  PR[91,3] = PR[90,3] + 26.195;
   1:  PR[92] = PR[91];
   1:  PR[92,3] = PR[92,3] + 20;
   1:J PR[92] 10% FINE;
   1:L PR[91] R[100]mm/sec CNT100;
   1:  CALL LASER_DRAHT_START;
   1:  PR[91,1] = PR[90,1] + 56.578;
   1:  PR[91,2] = PR[90,2] + 11.493;
   1:L PR[91] R[100]mm/sec CNT100;
   1:  PR[91,1] = PR[90,1] + 55.757;
   1:  PR[91,2] = PR[90,2] + 10.310;
   1:L PR[91] R[100]mm/sec CNT100;
   1:  PR[91,1] = PR[90,1] + 53.974;
   1:  PR[91,2] = PR[90,2] + 7.827;
   1:L PR[91] R[100]mm/sec CNT100;
   1:  PR[91,1] = PR[90,1] + 52.340;
   1:  PR[91,2] = PR[90,2] + 3.681;
   1:L PR[91] R[100]mm/sec CNT100;
   1:  PR[91,1] = PR[90,1] + 52.290;
   1:  PR[91,2] = PR[90,2] + 3.287;
   1:L PR[91] R[100]mm/sec CNT100;
   1:  PR[91,1] = PR[90,1] + 52.250;
   1:  PR[91,2] = PR[90,2] + 2.641;
   1:L PR[91] R[100]mm/sec CNT100;
   1:  PR[91,1] = PR[90,1] + 51.813;
   1:  PR[91,2] = PR[90,2] + -0.787;
   1:L PR[91] R[100]mm/sec CNT100;
   1:  PR[91,1] = PR[90,1] + 51.829;
   1:  PR[91,2] = PR[90,2] + -1.013;
   1:L PR[91] R[100]mm/sec CNT100;
   1:  PR[91,1] = PR[90,1] + 52.341;
   1:  PR[91,2] = PR[90,2] + -5.143;
   1:L PR[91] R[100]mm/sec CNT100;
   1:  PR[91,1] = PR[90,1] + 53.979;
   1:  PR[91,2] = PR[90,2] + -9.300;
   1:L PR[91] R[100]mm/sec CNT100;
   1:  PR[91,1] = PR[90,1] + 54.599;
   1:  PR[91,2] = PR[90,2] + -10.189;
   1:L PR[91] R[100]mm/sec CNT100;
   1:  PR[91,1] = PR[90,1] + 56.578;
   1:  PR[91,2] = PR[90,2] + -12.957;
   1:L PR[91] R[100]mm/sec CNT100;
   1:  PR[91,1] = PR[90,1] + 57.989;
   1:  PR[91,2] = PR[90,2] + -14.220;
   1:L PR[91] R[100]mm/sec CNT100;
   1:  PR[91,1] = PR[90,1] + 59.963;
   1:  PR[91,2] = PR[90,2] + -15.936;
   1:L PR[91] R[100]mm/sec CNT100;
   1:  PR[91,1] = PR[90,1] + 62.463;
   1:  PR[91,2] = PR[90,2] + -17.317;
   1:L PR[91] R[100]mm/sec CNT100;
   1:  PR[91,1] = PR[90,1] + 63.933;
   1:  PR[91,2] = PR[90,2] + -18.100;
   1:L PR[91] R[100]mm/sec CNT100;
   1:  PR[91,1] = PR[90,1] + 67.611;
   1:  PR[91,2] = PR[90,2] + -19.179;
   1:L PR[91] R[100]mm/sec CNT100;
   1:  PR[91,1] = PR[90,1] + 68.271;
   1:  PR[91,2] = PR[90,2] + -19.362;
   1:L PR[91] R[100]mm/sec CNT100;
   1:  PR[91,1] = PR[90,1] + 72.776;
   1:  PR[91,2] = PR[90,2] + -19.685;
   1:L PR[91] R[100]mm/sec CNT100;
   1:  PR[91,1] = PR[90,1] + 77.061;
   1:  PR[91,2] = PR[90,2] + -19.105;
   1:L PR[91] R[100]mm/sec CNT100;
   1:  PR[91,1] = PR[90,1] + 81.078;
   1:  PR[91,2] = PR[90,2] + -17.631;
   1:L PR[91] R[100]mm/sec CNT100;
   1:  PR[91,1] = PR[90,1] + 84.652;
   1:  PR[91,2] = PR[90,2] + -15.336;
   1:L PR[91] R[100]mm/sec CNT100;
   1:  PR[91,1] = PR[90,1] + 87.617;
   1:  PR[91,2] = PR[90,2] + -12.341;
   1:L PR[91] R[100]mm/sec CNT100;
   1:  PR[91,1] = PR[90,1] + 89.839;
   1:  PR[91,2] = PR[90,2] + -8.790;
   1:L PR[91] R[100]mm/sec CNT100;
   1:  PR[91,1] = PR[90,1] + 90.385;
   1:  PR[91,2] = PR[90,2] + -7.237;
   1:L PR[91] R[100]mm/sec CNT100;
   1:  PR[91,1] = PR[90,1] + 91.211;
   1:  PR[91,2] = PR[90,2] + -4.857;
   1:L PR[91] R[100]mm/sec CNT100;
   1:  PR[91,1] = PR[90,1] + 91.419;
   1:  PR[91,2] = PR[90,2] + -3.053;
   1:L PR[91] R[100]mm/sec CNT100;
   1:  PR[91,1] = PR[90,1] + 91.779;
   1:  PR[91,2] = PR[90,2] + -0.692;
   1:L PR[91] R[100]mm/sec CNT100;
   1:  PR[91,1] = PR[90,1] + 91.764;
   1:  PR[91,2] = PR[90,2] + -0.562;
   1:L PR[91] R[100]mm/sec CNT100;
   1:  PR[91,1] = PR[90,1] + 91.478;
   1:  PR[91,2] = PR[90,2] + 0.980;
   1:L PR[91] R[100]mm/sec CNT100;
   1:  PR[91,1] = PR[90,1] + 91.210;
   1:  PR[91,2] = PR[90,2] + 3.401;
   1:L PR[91] R[100]mm/sec CNT100;
   1:  PR[91,1] = PR[90,1] + 89.838;
   1:  PR[91,2] = PR[90,2] + 7.333;
   1:L PR[91] R[100]mm/sec CNT100;
   1:  PR[91,1] = PR[90,1] + 87.617;
   1:  PR[91,2] = PR[90,2] + 10.882;
   1:L PR[91] R[100]mm/sec CNT100;
   1:  PR[91,1] = PR[90,1] + 84.658;
   1:  PR[91,2] = PR[90,2] + 13.872;
   1:L PR[91] R[100]mm/sec CNT100;
   1:  PR[91,1] = PR[90,1] + 83.729;
   1:  PR[91,2] = PR[90,2] + 14.458;
   1:L PR[91] R[100]mm/sec CNT100;
   1:  PR[91,1] = PR[90,1] + 81.076;
   1:  PR[91,2] = PR[90,2] + 16.173;
   1:L PR[91] R[100]mm/sec CNT100;
   1:  PR[91,1] = PR[90,1] + 77.061;
   1:  PR[91,2] = PR[90,2] + 17.647;
   1:L PR[91] R[100]mm/sec CNT100;
   1:  PR[91,1] = PR[90,1] + 72.779;
   1:  PR[91,2] = PR[90,2] + 18.226;
   1:L PR[91] R[100]mm/sec CNT100;
   1:  PR[91,1] = PR[90,1] + 68.646;
   1:  PR[91,2] = PR[90,2] + 17.919;
   1:L PR[91] R[100]mm/sec CNT100;
   1:  PR[91,1] = PR[90,1] + 68.271;
   1:  PR[91,2] = PR[90,2] + 17.899;
   1:L PR[91] R[100]mm/sec CNT100;
   1:  PR[91,1] = PR[90,1] + 64.923;
   1:  PR[91,2] = PR[90,2] + 16.906;
   1:L PR[91] R[100]mm/sec CNT100;
   1:  PR[91,1] = PR[90,1] + 63.934;
   1:  PR[91,2] = PR[90,2] + 16.636;
   1:L PR[91] R[100]mm/sec CNT100;
   1:  PR[91,1] = PR[90,1] + 61.478;
   1:  PR[91,2] = PR[90,2] + 15.271;
   1:L PR[91] R[100]mm/sec CNT100;
   1:  PR[91,1] = PR[90,1] + 59.964;
   1:  PR[91,2] = PR[90,2] + 14.472;
   1:L PR[91] R[100]mm/sec CNT100;
   1:  PR[91,1] = PR[90,1] + 58.395;
   1:  PR[91,2] = PR[90,2] + 13.062;
   1:L PR[91] R[100]mm/sec CNT100TB   .50sec,CALL END_PUD;
   1:  PR[92] = PR[91];
   1:  PR[92,3] = PR[92,3] + 20;
   1:J PR[92] 10% FINE;
   1:  PR[91,1] = PR[90,1] + 41.160;
   1:  PR[91,2] = PR[90,2] + 8.184;
   1:  PR[92] = PR[91];
   1:  PR[92,3] = PR[92,3] + 20;
   1:J PR[92] 10% FINE;
   1:L PR[91] R[100]mm/sec CNT100;
   1:  CALL LASER_DRAHT_START;
   1:  PR[91,1] = PR[90,1] + 40.947;
   1:  PR[91,2] = PR[90,2] + 8.666;
   1:L PR[91] R[100]mm/sec CNT100;
   1:  PR[91,1] = PR[90,1] + 38.341;
   1:  PR[91,2] = PR[90,2] + 12.079;
   1:L PR[91] R[100]mm/sec CNT100;
   1:  PR[91,1] = PR[90,1] + 37.898;
   1:  PR[91,2] = PR[90,2] + 12.643;
   1:L PR[91] R[100]mm/sec CNT100;
   1:  PR[91,1] = PR[90,1] + 33.979;
   1:  PR[91,2] = PR[90,2] + 15.652;
   1:L PR[91] R[100]mm/sec CNT100;
   1:  PR[91,1] = PR[90,1] + 30.208;
   1:  PR[91,2] = PR[90,2] + 17.229;
   1:L PR[91] R[100]mm/sec CNT100;
   1:  PR[91,1] = PR[90,1] + 29.432;
   1:  PR[91,2] = PR[90,2] + 17.545;
   1:L PR[91] R[100]mm/sec CNT100;
   1:  PR[91,1] = PR[90,1] + 24.528;
   1:  PR[91,2] = PR[90,2] + 18.204;
   1:L PR[91] R[100]mm/sec CNT100;
   1:  PR[91,1] = PR[90,1] + 19.621;
   1:  PR[91,2] = PR[90,2] + 17.571;
   1:L PR[91] R[100]mm/sec CNT100;
   1:  PR[91,1] = PR[90,1] + 16.027;
   1:  PR[91,2] = PR[90,2] + 16.100;
   1:L PR[91] R[100]mm/sec CNT100;
   1:  PR[91,1] = PR[90,1] + 15.045;
   1:  PR[91,2] = PR[90,2] + 15.693;
   1:L PR[91] R[100]mm/sec CNT100;
   1:  PR[91,1] = PR[90,1] + 11.102;
   1:  PR[91,2] = PR[90,2] + 12.688;
   1:L PR[91] R[100]mm/sec CNT100;
   1:  PR[91,1] = PR[90,1] + 8.076;
   1:  PR[91,2] = PR[90,2] + 8.763;
   1:L PR[91] R[100]mm/sec CNT100;
   1:  PR[91,1] = PR[90,1] + 6.171;
   1:  PR[91,2] = PR[90,2] + 4.186;
   1:L PR[91] R[100]mm/sec CNT100;
   1:  PR[91,1] = PR[90,1] + 5.520;
   1:  PR[91,2] = PR[90,2] + -0.729;
   1:L PR[91] R[100]mm/sec CNT100;
   1:  PR[91,1] = PR[90,1] + 6.171;
   1:  PR[91,2] = PR[90,2] + -5.646;
   1:L PR[91] R[100]mm/sec CNT100;
   1:  PR[91,1] = PR[90,1] + 8.077;
   1:  PR[91,2] = PR[90,2] + -10.225;
   1:L PR[91] R[100]mm/sec CNT100;
   1:  PR[91,1] = PR[90,1] + 11.105;
   1:  PR[91,2] = PR[90,2] + -14.150;
   1:L PR[91] R[100]mm/sec CNT100;
   1:  PR[91,1] = PR[90,1] + 15.047;
   1:  PR[91,2] = PR[90,2] + -17.153;
   1:L PR[91] R[100]mm/sec CNT100;
   1:  PR[91,1] = PR[90,1] + 19.631;
   1:  PR[91,2] = PR[90,2] + -19.033;
   1:L PR[91] R[100]mm/sec CNT100;
   1:  PR[91,1] = PR[90,1] + 20.613;
   1:  PR[91,2] = PR[90,2] + -19.162;
   1:L PR[91] R[100]mm/sec CNT100;
   1:  PR[91,1] = PR[90,1] + 24.534;
   1:  PR[91,2] = PR[90,2] + -19.663;
   1:L PR[91] R[100]mm/sec CNT100;
   1:  PR[91,1] = PR[90,1] + 29.431;
   1:  PR[91,2] = PR[90,2] + -19.003;
   1:L PR[91] R[100]mm/sec CNT100;
   1:  PR[91,1] = PR[90,1] + 33.994;
   1:  PR[91,2] = PR[90,2] + -17.103;
   1:L PR[91] R[100]mm/sec CNT100;
   1:  PR[91,1] = PR[90,1] + 34.610;
   1:  PR[91,2] = PR[90,2] + -16.637;
   1:L PR[91] R[100]mm/sec CNT100;
   1:  PR[91,1] = PR[90,1] + 37.894;
   1:  PR[91,2] = PR[90,2] + -14.104;
   1:L PR[91] R[100]mm/sec CNT100;
   1:  PR[91,1] = PR[90,1] + 40.936;
   1:  PR[91,2] = PR[90,2] + -10.139;
   1:L PR[91] R[100]mm/sec CNT100;
   1:  PR[91,1] = PR[90,1] + 42.580;
   1:  PR[91,2] = PR[90,2] + -6.157;
   1:L PR[91] R[100]mm/sec CNT100;
   1:  PR[91,1] = PR[90,1] + 42.727;
   1:  PR[91,2] = PR[90,2] + -5.828;
   1:L PR[91] R[100]mm/sec CNT100;
   1:  PR[91,1] = PR[90,1] + 42.869;
   1:  PR[91,2] = PR[90,2] + -5.270;
   1:L PR[91] R[100]mm/sec CNT100;
   1:  PR[91,1] = PR[90,1] + 43.360;
   1:  PR[91,2] = PR[90,2] + -1.542;
   1:L PR[91] R[100]mm/sec CNT100;
   1:  PR[91,1] = PR[90,1] + 43.428;
   1:  PR[91,2] = PR[90,2] + -0.772;
   1:L PR[91] R[100]mm/sec CNT100;
   1:  PR[91,1] = PR[90,1] + 42.958;
   1:  PR[91,2] = PR[90,2] + 2.798;
   1:L PR[91] R[100]mm/sec CNT100;
   1:  PR[91,1] = PR[90,1] + 42.866;
   1:  PR[91,2] = PR[90,2] + 3.815;
   1:L PR[91] R[100]mm/sec CNT100;
   1:  PR[91,1] = PR[90,1] + 42.702;
   1:  PR[91,2] = PR[90,2] + 4.446;
   1:L PR[91] R[100]mm/sec CNT100;
   1:  PR[91,1] = PR[90,1] + 41.160;
   1:  PR[91,2] = PR[90,2] + 8.184;
   1:L PR[91] R[100]mm/sec CNT100TB   .50sec,CALL END_PUD;
   1:  PR[92] = PR[91];
   1:  PR[92,3] = PR[92,3] + 20;
   1:J PR[92] 10% FINE;
   1:  PR[91,1] = PR[90,1] + -27.836;
   1:  PR[91,2] = PR[90,2] + -18.849;
   1:  PR[92] = PR[91];
   1:  PR[92,3] = PR[92,3] + 20;
   1:J PR[92] 10% FINE;
   1:L PR[91] R[100]mm/sec CNT100;
   1:  CALL LASER_DRAHT_START;
   1:  PR[91,1] = PR[90,1] + -25.440;
   1:  PR[91,2] = PR[90,2] + -19.136;
   1:L PR[91] R[100]mm/sec CNT100;
   1:  PR[91,1] = PR[90,1] + -23.651;
   1:  PR[91,2] = PR[90,2] + -19.368;
   1:L PR[91] R[100]mm/sec CNT100;
   1:  PR[91,1] = PR[90,1] + -21.486;
   1:  PR[91,2] = PR[90,2] + -19.143;
   1:L PR[91] R[100]mm/sec CNT100;
   1:  PR[91,1] = PR[90,1] + -19.442;
   1:  PR[91,2] = PR[90,2] + -18.953;
   1:L PR[91] R[100]mm/sec CNT100;
   1:  PR[91,1] = PR[90,1] + -17.618;
   1:  PR[91,2] = PR[90,2] + -18.338;
   1:L PR[91] R[100]mm/sec CNT100;
   1:  PR[91,1] = PR[90,1] + -15.419;
   1:  PR[91,2] = PR[90,2] + -17.622;
   1:L PR[91] R[100]mm/sec CNT100;
   1:  PR[91,1] = PR[90,1] + -13.998;
   1:  PR[91,2] = PR[90,2] + -16.752;
   1:L PR[91] R[100]mm/sec CNT100;
   1:  PR[91,1] = PR[90,1] + -11.783;
   1:  PR[91,2] = PR[90,2] + -15.426;
   1:L PR[91] R[100]mm/sec CNT100;
   1:  PR[91,1] = PR[90,1] + -8.736;
   1:  PR[91,2] = PR[90,2] + -12.480;
   1:L PR[91] R[100]mm/sec CNT100;
   1:  PR[91,1] = PR[90,1] + -6.429;
   1:  PR[91,2] = PR[90,2] + -8.922;
   1:L PR[91] R[100]mm/sec CNT100;
   1:  PR[91,1] = PR[90,1] + -4.997;
   1:  PR[91,2] = PR[90,2] + -4.946;
   1:L PR[91] R[100]mm/sec CNT100;
   1:  PR[91,1] = PR[90,1] + -4.548;
   1:  PR[91,2] = PR[90,2] + -0.738;
   1:L PR[91] R[100]mm/sec CNT100;
   1:  PR[91,1] = PR[90,1] + -4.635;
   1:  PR[91,2] = PR[90,2] + 0.012;
   1:L PR[91] R[100]mm/sec CNT100;
   1:  PR[91,1] = PR[90,1] + -4.624;
   1:  PR[91,2] = PR[90,2] + 0.292;
   1:L PR[91] R[100]mm/sec CNT100;
   1:  PR[91,1] = PR[90,1] + -4.994;
   1:  PR[91,2] = PR[90,2] + 3.478;
   1:L PR[91] R[100]mm/sec CNT100;
   1:  PR[91,1] = PR[90,1] + -6.429;
   1:  PR[91,2] = PR[90,2] + 7.463;
   1:L PR[91] R[100]mm/sec CNT100;
   1:  PR[91,1] = PR[90,1] + -8.736;
   1:  PR[91,2] = PR[90,2] + 11.021;
   1:L PR[91] R[100]mm/sec CNT100;
   1:  PR[91,1] = PR[90,1] + -11.790;
   1:  PR[91,2] = PR[90,2] + 13.974;
   1:L PR[91] R[100]mm/sec CNT100;
   1:  PR[91,1] = PR[90,1] + -13.095;
   1:  PR[91,2] = PR[90,2] + 14.772;
   1:L PR[91] R[100]mm/sec CNT100;
   1:  PR[91,1] = PR[90,1] + -15.419;
   1:  PR[91,2] = PR[90,2] + 16.165;
   1:L PR[91] R[100]mm/sec CNT100;
   1:  PR[91,1] = PR[90,1] + -17.136;
   1:  PR[91,2] = PR[90,2] + 16.744;
   1:L PR[91] R[100]mm/sec CNT100;
   1:  PR[91,1] = PR[90,1] + -19.442;
   1:  PR[91,2] = PR[90,2] + 17.497;
   1:L PR[91] R[100]mm/sec CNT100;
   1:  PR[91,1] = PR[90,1] + -21.527;
   1:  PR[91,2] = PR[90,2] + 17.713;
   1:L PR[91] R[100]mm/sec CNT100;
   1:  PR[91,1] = PR[90,1] + -23.651;
   1:  PR[91,2] = PR[90,2] + 17.912;
   1:L PR[91] R[100]mm/sec CNT100;
   1:  PR[91,1] = PR[90,1] + -25.996;
   1:  PR[91,2] = PR[90,2] + 17.631;
   1:L PR[91] R[100]mm/sec CNT100;
   1:  PR[91,1] = PR[90,1] + -27.833;
   1:  PR[91,2] = PR[90,2] + 17.393;
   1:L PR[91] R[100]mm/sec CNT100;
   1:  PR[91,1] = PR[90,1] + -31.795;
   1:  PR[91,2] = PR[90,2] + 15.974;
   1:L PR[91] R[100]mm/sec CNT100;
   1:  PR[91,1] = PR[90,1] + -34.157;
   1:  PR[91,2] = PR[90,2] + 14.483;
   1:L PR[91] R[100]mm/sec CNT100;
   1:  PR[91,1] = PR[90,1] + -35.320;
   1:  PR[91,2] = PR[90,2] + 13.736;
   1:L PR[91] R[100]mm/sec CNT100;
   1:  PR[91,1] = PR[90,1] + -38.261;
   1:  PR[91,2] = PR[90,2] + 10.783;
   1:L PR[91] R[100]mm/sec CNT100;
   1:  PR[91,1] = PR[90,1] + -40.465;
   1:  PR[91,2] = PR[90,2] + 7.271;
   1:L PR[91] R[100]mm/sec CNT100;
   1:  PR[91,1] = PR[90,1] + -41.829;
   1:  PR[91,2] = PR[90,2] + 3.370;
   1:L PR[91] R[100]mm/sec CNT100;
   1:  PR[91,1] = PR[90,1] + -42.198;
   1:  PR[91,2] = PR[90,2] + 0.121;
   1:L PR[91] R[100]mm/sec CNT100;
   1:  PR[91,1] = PR[90,1] + -42.279;
   1:  PR[91,2] = PR[90,2] + -0.278;
   1:L PR[91] R[100]mm/sec CNT100;
   1:  PR[91,1] = PR[90,1] + -42.329;
   1:  PR[91,2] = PR[90,2] + -0.717;
   1:L PR[91] R[100]mm/sec CNT100;
   1:  PR[91,1] = PR[90,1] + -41.936;
   1:  PR[91,2] = PR[90,2] + -3.871;
   1:L PR[91] R[100]mm/sec CNT100;
   1:  PR[91,1] = PR[90,1] + -41.829;
   1:  PR[91,2] = PR[90,2] + -4.830;
   1:L PR[91] R[100]mm/sec CNT100;
   1:  PR[91,1] = PR[90,1] + -40.465;
   1:  PR[91,2] = PR[90,2] + -8.730;
   1:L PR[91] R[100]mm/sec CNT100;
   1:  PR[91,1] = PR[90,1] + -38.261;
   1:  PR[91,2] = PR[90,2] + -12.242;
   1:L PR[91] R[100]mm/sec CNT100;
   1:  PR[91,1] = PR[90,1] + -35.324;
   1:  PR[91,2] = PR[90,2] + -15.192;
   1:L PR[91] R[100]mm/sec CNT100;
   1:  PR[91,1] = PR[90,1] + -31.796;
   1:  PR[91,2] = PR[90,2] + -17.431;
   1:L PR[91] R[100]mm/sec CNT100;
   1:  PR[91,1] = PR[90,1] + -29.320;
   1:  PR[91,2] = PR[90,2] + -18.308;
   1:L PR[91] R[100]mm/sec CNT100;
   1:  PR[91,1] = PR[90,1] + -27.836;
   1:  PR[91,2] = PR[90,2] + -18.849;
   1:L PR[91] R[100]mm/sec CNT100TB   .50sec,CALL END_PUD;
   1:  PR[92] = PR[91];
   1:  PR[92,3] = PR[92,3] + 20;
   1:J PR[92] 10% FINE;
   1:  PR[91,1] = PR[90,1] + -59.903;
   1:  PR[91,2] = PR[90,2] + 13.243;
   1:  PR[92] = PR[91];
   1:  PR[92,3] = PR[92,3] + 20;
   1:J PR[92] 10% FINE;
   1:L PR[91] R[100]mm/sec CNT100;
   1:  CALL LASER_DRAHT_START;
   1:  PR[91,1] = PR[90,1] + -63.277;
   1:  PR[91,2] = PR[90,2] + 15.489;
   1:L PR[91] R[100]mm/sec CNT100;
   1:  PR[91,1] = PR[90,1] + -67.051;
   1:  PR[91,2] = PR[90,2] + 17.006;
   1:L PR[91] R[100]mm/sec CNT100;
   1:  PR[91,1] = PR[90,1] + -71.057;
   1:  PR[91,2] = PR[90,2] + 17.738;
   1:L PR[91] R[100]mm/sec CNT100;
   1:  PR[91,1] = PR[90,1] + -75.056;
   1:  PR[91,2] = PR[90,2] + 17.673;
   1:L PR[91] R[100]mm/sec CNT100;
   1:  PR[91,1] = PR[90,1] + -78.887;
   1:  PR[91,2] = PR[90,2] + 16.820;
   1:L PR[91] R[100]mm/sec CNT100;
   1:  PR[91,1] = PR[90,1] + -82.443;
   1:  PR[91,2] = PR[90,2] + 15.213;
   1:L PR[91] R[100]mm/sec CNT100;
   1:  PR[91,1] = PR[90,1] + -85.580;
   1:  PR[91,2] = PR[90,2] + 12.923;
   1:L PR[91] R[100]mm/sec CNT100;
   1:  PR[91,1] = PR[90,1] + -88.164;
   1:  PR[91,2] = PR[90,2] + 10.051;
   1:L PR[91] R[100]mm/sec CNT100;
   1:  PR[91,1] = PR[90,1] + -90.091;
   1:  PR[91,2] = PR[90,2] + 6.722;
   1:L PR[91] R[100]mm/sec CNT100;
   1:  PR[91,1] = PR[90,1] + -91.279;
   1:  PR[91,2] = PR[90,2] + 3.075;
   1:L PR[91] R[100]mm/sec CNT100;
   1:  PR[91,1] = PR[90,1] + -91.449;
   1:  PR[91,2] = PR[90,2] + 1.478;
   1:L PR[91] R[100]mm/sec CNT100;
   1:  PR[91,1] = PR[90,1] + -91.504;
   1:  PR[91,2] = PR[90,2] + 1.218;
   1:L PR[91] R[100]mm/sec CNT100;
   1:  PR[91,1] = PR[90,1] + -91.792;
   1:  PR[91,2] = PR[90,2] + -0.720;
   1:L PR[91] R[100]mm/sec CNT100;
   1:  PR[91,1] = PR[90,1] + -91.545;
   1:  PR[91,2] = PR[90,2] + -2.284;
   1:L PR[91] R[100]mm/sec CNT100;
   1:  PR[91,1] = PR[90,1] + -91.428;
   1:  PR[91,2] = PR[90,2] + -2.781;
   1:L PR[91] R[100]mm/sec CNT100;
   1:  PR[91,1] = PR[90,1] + -91.245;
   1:  PR[91,2] = PR[90,2] + -4.536;
   1:L PR[91] R[100]mm/sec CNT100;
   1:  PR[91,1] = PR[90,1] + -90.580;
   1:  PR[91,2] = PR[90,2] + -6.563;
   1:L PR[91] R[100]mm/sec CNT100;
   1:  PR[91,1] = PR[90,1] + -90.054;
   1:  PR[91,2] = PR[90,2] + -8.183;
   1:L PR[91] R[100]mm/sec CNT100;
   1:  PR[91,1] = PR[90,1] + -88.122;
   1:  PR[91,2] = PR[90,2] + -11.513;
   1:L PR[91] R[100]mm/sec CNT100;
   1:  PR[91,1] = PR[90,1] + -85.530;
   1:  PR[91,2] = PR[90,2] + -14.388;
   1:L PR[91] R[100]mm/sec CNT100;
   1:  PR[91,1] = PR[90,1] + -82.382;
   1:  PR[91,2] = PR[90,2] + -16.682;
   1:L PR[91] R[100]mm/sec CNT100;
   1:  PR[91,1] = PR[90,1] + -78.812;
   1:  PR[91,2] = PR[90,2] + -18.295;
   1:L PR[91] R[100]mm/sec CNT100;
   1:  PR[91,1] = PR[90,1] + -74.967;
   1:  PR[91,2] = PR[90,2] + -19.151;
   1:L PR[91] R[100]mm/sec CNT100;
   1:  PR[91,1] = PR[90,1] + -71.014;
   1:  PR[91,2] = PR[90,2] + -19.210;
   1:L PR[91] R[100]mm/sec CNT100;
   1:  PR[91,1] = PR[90,1] + -67.120;
   1:  PR[91,2] = PR[90,2] + -18.462;
   1:L PR[91] R[100]mm/sec CNT100;
   1:  PR[91,1] = PR[90,1] + -65.650;
   1:  PR[91,2] = PR[90,2] + -17.846;
   1:L PR[91] R[100]mm/sec CNT100;
   1:  PR[91,1] = PR[90,1] + -63.333;
   1:  PR[91,2] = PR[90,2] + -16.929;
   1:L PR[91] R[100]mm/sec CNT100;
   1:  PR[91,1] = PR[90,1] + -59.926;
   1:  PR[91,2] = PR[90,2] + -14.691;
   1:L PR[91] R[100]mm/sec CNT100;
   1:  PR[91,1] = PR[90,1] + -57.766;
   1:  PR[91,2] = PR[90,2] + -12.491;
   1:L PR[91] R[100]mm/sec CNT100;
   1:  PR[91,1] = PR[90,1] + -57.074;
   1:  PR[91,2] = PR[90,2] + -11.805;
   1:L PR[91] R[100]mm/sec CNT100;
   1:  PR[91,1] = PR[90,1] + -55.664;
   1:  PR[91,2] = PR[90,2] + -9.558;
   1:L PR[91] R[100]mm/sec CNT100;
   1:  PR[91,1] = PR[90,1] + -54.929;
   1:  PR[91,2] = PR[90,2] + -8.413;
   1:L PR[91] R[100]mm/sec CNT100;
   1:  PR[91,1] = PR[90,1] + -53.599;
   1:  PR[91,2] = PR[90,2] + -4.666;
   1:L PR[91] R[100]mm/sec CNT100;
   1:  PR[91,1] = PR[90,1] + -53.360;
   1:  PR[91,2] = PR[90,2] + -2.607;
   1:L PR[91] R[100]mm/sec CNT100;
   1:  PR[91,1] = PR[90,1] + -53.225;
   1:  PR[91,2] = PR[90,2] + -0.745;
   1:L PR[91] R[100]mm/sec CNT100;
   1:  PR[91,1] = PR[90,1] + -53.308;
   1:  PR[91,2] = PR[90,2] + 0.189;
   1:L PR[91] R[100]mm/sec CNT100;
   1:  PR[91,1] = PR[90,1] + -53.649;
   1:  PR[91,2] = PR[90,2] + 3.212;
   1:L PR[91] R[100]mm/sec CNT100;
   1:  PR[91,1] = PR[90,1] + -54.966;
   1:  PR[91,2] = PR[90,2] + 6.966;
   1:L PR[91] R[100]mm/sec CNT100;
   1:  PR[91,1] = PR[90,1] + -57.088;
   1:  PR[91,2] = PR[90,2] + 10.361;
   1:L PR[91] R[100]mm/sec CNT100;
   1:  PR[91,1] = PR[90,1] + -59.903;
   1:  PR[91,2] = PR[90,2] + 13.243;
   1:L PR[91] R[100]mm/sec CNT100TB   .50sec,CALL END_PUD;
   1:  PR[92] = PR[91];
   1:  PR[92,3] = PR[92,3] + 20;
   1:J PR[92] 10% FINE;
   1:  PR[91] = PR[90];
   1:  PR[91,1] = PR[90,1] + 91.045;
   1:  PR[91,2] = PR[90,2] + 3.417;
   1:  PR[91,3] = PR[90,3] + 27.495;
   1:  PR[92] = PR[91];
   1:  PR[92,3] = PR[92,3] + 20;
   1:J PR[92] 10% FINE;
   1:L PR[91] R[100]mm/sec CNT100;
   1:  CALL LASER_DRAHT_START;
   1:  PR[91,1] = PR[90,1] + 89.670;
   1:  PR[91,2] = PR[90,2] + 7.365;
   1:L PR[91] R[100]mm/sec CNT100;
   1:  PR[91,1] = PR[90,1] + 87.443;
   1:  PR[91,2] = PR[90,2] + 10.931;
   1:L PR[91] R[100]mm/sec CNT100;
   1:  PR[91,1] = PR[90,1] + 84.468;
   1:  PR[91,2] = PR[90,2] + 13.943;
   1:L PR[91] R[100]mm/sec CNT100;
   1:  PR[91,1] = PR[90,1] + 80.881;
   1:  PR[91,2] = PR[90,2] + 16.252;
   1:L PR[91] R[100]mm/sec CNT100;
   1:  PR[91,1] = PR[90,1] + 76.821;
   1:  PR[91,2] = PR[90,2] + 17.748;
   1:L PR[91] R[100]mm/sec CNT100;
   1:  PR[91,1] = PR[90,1] + 72.793;
   1:  PR[91,2] = PR[90,2] + 18.312;
   1:L PR[91] R[100]mm/sec CNT100;
   1:  PR[91,1] = PR[90,1] + 72.358;
   1:  PR[91,2] = PR[90,2] + 18.382;
   1:L PR[91] R[100]mm/sec CNT100;
   1:  PR[91,1] = PR[90,1] + 68.913;
   1:  PR[91,2] = PR[90,2] + 18.126;
   1:L PR[91] R[100]mm/sec CNT100;
   1:  PR[91,1] = PR[90,1] + 67.834;
   1:  PR[91,2] = PR[90,2] + 18.069;
   1:L PR[91] R[100]mm/sec CNT100;
   1:  PR[91,1] = PR[90,1] + 65.170;
   1:  PR[91,2] = PR[90,2] + 17.279;
   1:L PR[91] R[100]mm/sec CNT100;
   1:  PR[91,1] = PR[90,1] + 63.449;
   1:  PR[91,2] = PR[90,2] + 16.811;
   1:L PR[91] R[100]mm/sec CNT100;
   1:  PR[91,1] = PR[90,1] + 61.667;
   1:  PR[91,2] = PR[90,2] + 15.820;
   1:L PR[91] R[100]mm/sec CNT100;
   1:  PR[91,1] = PR[90,1] + 59.428;
   1:  PR[91,2] = PR[90,2] + 14.638;
   1:L PR[91] R[100]mm/sec CNT100;
   1:  PR[91,1] = PR[90,1] + 58.480;
   1:  PR[91,2] = PR[90,2] + 13.786;
   1:L PR[91] R[100]mm/sec CNT100;
   1:  PR[91,1] = PR[90,1] + 55.992;
   1:  PR[91,2] = PR[90,2] + 11.637;
   1:L PR[91] R[100]mm/sec CNT100;
   1:  PR[91,1] = PR[90,1] + 55.687;
   1:  PR[91,2] = PR[90,2] + 11.198;
   1:L PR[91] R[100]mm/sec CNT100;
   1:  PR[91,1] = PR[90,1] + 53.343;
   1:  PR[91,2] = PR[90,2] + 7.934;
   1:L PR[91] R[100]mm/sec CNT100;
   1:  PR[91,1] = PR[90,1] + 52.852;
   1:  PR[91,2] = PR[90,2] + 6.692;
   1:L PR[91] R[100]mm/sec CNT100;
   1:  PR[91,1] = PR[90,1] + 51.596;
   1:  PR[91,2] = PR[90,2] + 3.729;
   1:L PR[91] R[100]mm/sec CNT100;
   1:  PR[91,1] = PR[90,1] + 51.566;
   1:  PR[91,2] = PR[90,2] + 3.532;
   1:L PR[91] R[100]mm/sec CNT100;
   1:  PR[91,1] = PR[90,1] + 50.974;
   1:  PR[91,2] = PR[90,2] + -0.729;
   1:L PR[91] R[100]mm/sec CNT100;
   1:  PR[91,1] = PR[90,1] + 51.566;
   1:  PR[91,2] = PR[90,2] + -4.991;
   1:L PR[91] R[100]mm/sec CNT100;
   1:  PR[91,1] = PR[90,1] + 51.596;
   1:  PR[91,2] = PR[90,2] + -5.188;
   1:L PR[91] R[100]mm/sec CNT100;
   1:  PR[91,1] = PR[90,1] + 52.852;
   1:  PR[91,2] = PR[90,2] + -8.151;
   1:L PR[91] R[100]mm/sec CNT100;
   1:  PR[91,1] = PR[90,1] + 53.344;
   1:  PR[91,2] = PR[90,2] + -9.395;
   1:L PR[91] R[100]mm/sec CNT100;
   1:  PR[91,1] = PR[90,1] + 55.992;
   1:  PR[91,2] = PR[90,2] + -13.102;
   1:L PR[91] R[100]mm/sec CNT100;
   1:  PR[91,1] = PR[90,1] + 56.547;
   1:  PR[91,2] = PR[90,2] + -13.598;
   1:L PR[91] R[100]mm/sec CNT100;
   1:  PR[91,1] = PR[90,1] + 59.428;
   1:  PR[91,2] = PR[90,2] + -16.102;
   1:L PR[91] R[100]mm/sec CNT100;
   1:  PR[91,1] = PR[90,1] + 60.964;
   1:  PR[91,2] = PR[90,2] + -16.951;
   1:L PR[91] R[100]mm/sec CNT100;
   1:  PR[91,1] = PR[90,1] + 63.449;
   1:  PR[91,2] = PR[90,2] + -18.274;
   1:L PR[91] R[100]mm/sec CNT100;
   1:  PR[91,1] = PR[90,1] + 66.138;
   1:  PR[91,2] = PR[90,2] + -19.063;
   1:L PR[91] R[100]mm/sec CNT100;
   1:  PR[91,1] = PR[90,1] + 67.834;
   1:  PR[91,2] = PR[90,2] + -19.532;
   1:L PR[91] R[100]mm/sec CNT100;
   1:  PR[91,1] = PR[90,1] + 71.592;
   1:  PR[91,2] = PR[90,2] + -19.801;
   1:L PR[91] R[100]mm/sec CNT100;
   1:  PR[91,1] = PR[90,1] + 72.358;
   1:  PR[91,2] = PR[90,2] + -19.844;
   1:L PR[91] R[100]mm/sec CNT100;
   1:  PR[91,1] = PR[90,1] + 76.818;
   1:  PR[91,2] = PR[90,2] + -19.208;
   1:L PR[91] R[100]mm/sec CNT100;
   1:  PR[91,1] = PR[90,1] + 80.881;
   1:  PR[91,2] = PR[90,2] + -17.711;
   1:L PR[91] R[100]mm/sec CNT100;
   1:  PR[91,1] = PR[90,1] + 84.468;
   1:  PR[91,2] = PR[90,2] + -15.401;
   1:L PR[91] R[100]mm/sec CNT100;
   1:  PR[91,1] = PR[90,1] + 87.446;
   1:  PR[91,2] = PR[90,2] + -12.387;
   1:L PR[91] R[100]mm/sec CNT100;
   1:  PR[91,1] = PR[90,1] + 87.928;
   1:  PR[91,2] = PR[90,2] + -11.623;
   1:L PR[91] R[100]mm/sec CNT100;
   1:  PR[91,1] = PR[90,1] + 89.669;
   1:  PR[91,2] = PR[90,2] + -8.826;
   1:L PR[91] R[100]mm/sec CNT100;
   1:  PR[91,1] = PR[90,1] + 91.047;
   1:  PR[91,2] = PR[90,2] + -4.872;
   1:L PR[91] R[100]mm/sec CNT100;
   1:  PR[91,1] = PR[90,1] + 91.193;
   1:  PR[91,2] = PR[90,2] + -3.604;
   1:L PR[91] R[100]mm/sec CNT100;
   1:  PR[91,1] = PR[90,1] + 91.572;
   1:  PR[91,2] = PR[90,2] + -1.114;
   1:L PR[91] R[100]mm/sec CNT100;
   1:  PR[91,1] = PR[90,1] + 91.607;
   1:  PR[91,2] = PR[90,2] + -0.801;
   1:L PR[91] R[100]mm/sec CNT100;
   1:  PR[91,1] = PR[90,1] + 91.372;
   1:  PR[91,2] = PR[90,2] + 0.468;
   1:L PR[91] R[100]mm/sec CNT100;
   1:  PR[91,1] = PR[90,1] + 91.045;
   1:  PR[91,2] = PR[90,2] + 3.417;
   1:L PR[91] R[100]mm/sec CNT100TB   .50sec,CALL END_PUD;
   1:  PR[92] = PR[91];
   1:  PR[92,3] = PR[92,3] + 20;
   1:J PR[92] 10% FINE;
   1:  PR[91,1] = PR[90,1] + 24.459;
   1:  PR[91,2] = PR[90,2] + -19.805;
   1:  PR[92] = PR[91];
   1:  PR[92,3] = PR[92,3] + 20;
   1:J PR[92] 10% FINE;
   1:L PR[91] R[100]mm/sec CNT100;
   1:  CALL LASER_DRAHT_START;
   1:  PR[91,1] = PR[90,1] + 29.392;
   1:  PR[91,2] = PR[90,2] + -19.144;
   1:L PR[91] R[100]mm/sec CNT100;
   1:  PR[91,1] = PR[90,1] + 33.986;
   1:  PR[91,2] = PR[90,2] + -17.234;
   1:L PR[91] R[100]mm/sec CNT100;
   1:  PR[91,1] = PR[90,1] + 34.996;
   1:  PR[91,2] = PR[90,2] + -16.469;
   1:L PR[91] R[100]mm/sec CNT100;
   1:  PR[91,1] = PR[90,1] + 37.921;
   1:  PR[91,2] = PR[90,2] + -14.213;
   1:L PR[91] R[100]mm/sec CNT100;
   1:  PR[91,1] = PR[90,1] + 38.674;
   1:  PR[91,2] = PR[90,2] + -13.250;
   1:L PR[91] R[100]mm/sec CNT100;
   1:  PR[91,1] = PR[90,1] + 41.002;
   1:  PR[91,2] = PR[90,2] + -10.202;
   1:L PR[91] R[100]mm/sec CNT100;
   1:  PR[91,1] = PR[90,1] + 41.006;
   1:  PR[91,2] = PR[90,2] + -10.195;
   1:L PR[91] R[100]mm/sec CNT100;
   1:  PR[91,1] = PR[90,1] + 42.478;
   1:  PR[91,2] = PR[90,2] + -6.631;
   1:L PR[91] R[100]mm/sec CNT100;
   1:  PR[91,1] = PR[90,1] + 42.735;
   1:  PR[91,2] = PR[90,2] + -6.057;
   1:L PR[91] R[100]mm/sec CNT100;
   1:  PR[91,1] = PR[90,1] + 42.992;
   1:  PR[91,2] = PR[90,2] + -5.050;
   1:L PR[91] R[100]mm/sec CNT100;
   1:  PR[91,1] = PR[90,1] + 43.381;
   1:  PR[91,2] = PR[90,2] + -2.091;
   1:L PR[91] R[100]mm/sec CNT100;
   1:  PR[91,1] = PR[90,1] + 43.498;
   1:  PR[91,2] = PR[90,2] + -0.772;
   1:L PR[91] R[100]mm/sec CNT100;
   1:  PR[91,1] = PR[90,1] + 43.139;
   1:  PR[91,2] = PR[90,2] + 1.951;
   1:L PR[91] R[100]mm/sec CNT100;
   1:  PR[91,1] = PR[90,1] + 42.991;
   1:  PR[91,2] = PR[90,2] + 3.577;
   1:L PR[91] R[100]mm/sec CNT100;
   1:  PR[91,1] = PR[90,1] + 42.700;
   1:  PR[91,2] = PR[90,2] + 4.702;
   1:L PR[91] R[100]mm/sec CNT100;
   1:  PR[91,1] = PR[90,1] + 41.393;
   1:  PR[91,2] = PR[90,2] + 7.870;
   1:L PR[91] R[100]mm/sec CNT100;
   1:  PR[91,1] = PR[90,1] + 41.029;
   1:  PR[91,2] = PR[90,2] + 8.694;
   1:L PR[91] R[100]mm/sec CNT100;
   1:  PR[91,1] = PR[90,1] + 41.002;
   1:  PR[91,2] = PR[90,2] + 8.744;
   1:L PR[91] R[100]mm/sec CNT100;
   1:  PR[91,1] = PR[90,1] + 38.663;
   1:  PR[91,2] = PR[90,2] + 11.810;
   1:L PR[91] R[100]mm/sec CNT100;
   1:  PR[91,1] = PR[90,1] + 37.914;
   1:  PR[91,2] = PR[90,2] + 12.762;
   1:L PR[91] R[100]mm/sec CNT100;
   1:  PR[91,1] = PR[90,1] + 34.989;
   1:  PR[91,2] = PR[90,2] + 15.018;
   1:L PR[91] R[100]mm/sec CNT100;
   1:  PR[91,1] = PR[90,1] + 33.975;
   1:  PR[91,2] = PR[90,2] + 15.782;
   1:L PR[91] R[100]mm/sec CNT100;
   1:  PR[91,1] = PR[90,1] + 30.626;
   1:  PR[91,2] = PR[90,2] + 17.182;
   1:L PR[91] R[100]mm/sec CNT100;
   1:  PR[91,1] = PR[90,1] + 29.388;
   1:  PR[91,2] = PR[90,2] + 17.687;
   1:L PR[91] R[100]mm/sec CNT100;
   1:  PR[91,1] = PR[90,1] + 24.450;
   1:  PR[91,2] = PR[90,2] + 18.346;
   1:L PR[91] R[100]mm/sec CNT100;
   1:  PR[91,1] = PR[90,1] + 19.510;
   1:  PR[91,2] = PR[90,2] + 17.707;
   1:L PR[91] R[100]mm/sec CNT100;
   1:  PR[91,1] = PR[90,1] + 16.366;
   1:  PR[91,2] = PR[90,2] + 16.420;
   1:L PR[91] R[100]mm/sec CNT100;
   1:  PR[91,1] = PR[90,1] + 14.901;
   1:  PR[91,2] = PR[90,2] + 15.814;
   1:L PR[91] R[100]mm/sec CNT100;
   1:  PR[91,1] = PR[90,1] + 10.931;
   1:  PR[91,2] = PR[90,2] + 12.787;
   1:L PR[91] R[100]mm/sec CNT100;
   1:  PR[91,1] = PR[90,1] + 7.883;
   1:  PR[91,2] = PR[90,2] + 8.833;
   1:L PR[91] R[100]mm/sec CNT100;
   1:  PR[91,1] = PR[90,1] + 6.643;
   1:  PR[91,2] = PR[90,2] + 5.854;
   1:L PR[91] R[100]mm/sec CNT100;
   1:  PR[91,1] = PR[90,1] + 5.965;
   1:  PR[91,2] = PR[90,2] + 4.223;
   1:L PR[91] R[100]mm/sec CNT100;
   1:  PR[91,1] = PR[90,1] + 5.310;
   1:  PR[91,2] = PR[90,2] + -0.729;
   1:L PR[91] R[100]mm/sec CNT100;
   1:  PR[91,1] = PR[90,1] + 5.965;
   1:  PR[91,2] = PR[90,2] + -5.683;
   1:L PR[91] R[100]mm/sec CNT100;
   1:  PR[91,1] = PR[90,1] + 7.885;
   1:  PR[91,2] = PR[90,2] + -10.295;
   1:L PR[91] R[100]mm/sec CNT100;
   1:  PR[91,1] = PR[90,1] + 8.936;
   1:  PR[91,2] = PR[90,2] + -11.660;
   1:L PR[91] R[100]mm/sec CNT100;
   1:  PR[91,1] = PR[90,1] + 10.935;
   1:  PR[91,2] = PR[90,2] + -14.249;
   1:L PR[91] R[100]mm/sec CNT100;
   1:  PR[91,1] = PR[90,1] + 14.905;
   1:  PR[91,2] = PR[90,2] + -17.275;
   1:L PR[91] R[100]mm/sec CNT100;
   1:  PR[91,1] = PR[90,1] + 19.521;
   1:  PR[91,2] = PR[90,2] + -19.169;
   1:L PR[91] R[100]mm/sec CNT100;
   1:  PR[91,1] = PR[90,1] + 21.012;
   1:  PR[91,2] = PR[90,2] + -19.365;
   1:L PR[91] R[100]mm/sec CNT100;
   1:  PR[91,1] = PR[90,1] + 24.459;
   1:  PR[91,2] = PR[90,2] + -19.805;
   1:L PR[91] R[100]mm/sec CNT100TB   .50sec,CALL END_PUD;
   1:  PR[92] = PR[91];
   1:  PR[92,3] = PR[92,3] + 20;
   1:J PR[92] 10% FINE;
   1:  PR[91,1] = PR[90,1] + -12.346;
   1:  PR[91,2] = PR[90,2] + 14.551;
   1:  PR[92] = PR[91];
   1:  PR[92,3] = PR[92,3] + 20;
   1:J PR[92] 10% FINE;
   1:L PR[91] R[100]mm/sec CNT100;
   1:  CALL LASER_DRAHT_START;
   1:  PR[91,1] = PR[90,1] + -15.179;
   1:  PR[91,2] = PR[90,2] + 16.250;
   1:L PR[91] R[100]mm/sec CNT100;
   1:  PR[91,1] = PR[90,1] + -19.233;
   1:  PR[91,2] = PR[90,2] + 17.587;
   1:L PR[91] R[100]mm/sec CNT100;
   1:  PR[91,1] = PR[90,1] + -20.779;
   1:  PR[91,2] = PR[90,2] + 17.747;
   1:L PR[91] R[100]mm/sec CNT100;
   1:  PR[91,1] = PR[90,1] + -23.460;
   1:  PR[91,2] = PR[90,2] + 17.998;
   1:L PR[91] R[100]mm/sec CNT100;
   1:  PR[91,1] = PR[90,1] + -25.292;
   1:  PR[91,2] = PR[90,2] + 17.779;
   1:L PR[91] R[100]mm/sec CNT100;
   1:  PR[91,1] = PR[90,1] + -27.663;
   1:  PR[91,2] = PR[90,2] + 17.472;
   1:L PR[91] R[100]mm/sec CNT100;
   1:  PR[91,1] = PR[90,1] + -29.647;
   1:  PR[91,2] = PR[90,2] + 16.769;
   1:L PR[91] R[100]mm/sec CNT100;
   1:  PR[91,1] = PR[90,1] + -31.633;
   1:  PR[91,2] = PR[90,2] + 16.046;
   1:L PR[91] R[100]mm/sec CNT100;
   1:  PR[91,1] = PR[90,1] + -33.599;
   1:  PR[91,2] = PR[90,2] + 14.805;
   1:L PR[91] R[100]mm/sec CNT100;
   1:  PR[91,1] = PR[90,1] + -35.174;
   1:  PR[91,2] = PR[90,2] + 13.794;
   1:L PR[91] R[100]mm/sec CNT100;
   1:  PR[91,1] = PR[90,1] + -38.124;
   1:  PR[91,2] = PR[90,2] + 10.827;
   1:L PR[91] R[100]mm/sec CNT100;
   1:  PR[91,1] = PR[90,1] + -40.335;
   1:  PR[91,2] = PR[90,2] + 7.301;
   1:L PR[91] R[100]mm/sec CNT100;
   1:  PR[91,1] = PR[90,1] + -41.703;
   1:  PR[91,2] = PR[90,2] + 3.385;
   1:L PR[91] R[100]mm/sec CNT100;
   1:  PR[91,1] = PR[90,1] + -42.024;
   1:  PR[91,2] = PR[90,2] + 0.555;
   1:L PR[91] R[100]mm/sec CNT100;
   1:  PR[91,1] = PR[90,1] + -42.096;
   1:  PR[91,2] = PR[90,2] + 0.206;
   1:L PR[91] R[100]mm/sec CNT100;
   1:  PR[91,1] = PR[90,1] + -42.199;
   1:  PR[91,2] = PR[90,2] + -0.717;
   1:L PR[91] R[100]mm/sec CNT100;
   1:  PR[91,1] = PR[90,1] + -41.858;
   1:  PR[91,2] = PR[90,2] + -3.458;
   1:L PR[91] R[100]mm/sec CNT100;
   1:  PR[91,1] = PR[90,1] + -41.703;
   1:  PR[91,2] = PR[90,2] + -4.845;
   1:L PR[91] R[100]mm/sec CNT100;
   1:  PR[91,1] = PR[90,1] + -40.335;
   1:  PR[91,2] = PR[90,2] + -8.760;
   1:L PR[91] R[100]mm/sec CNT100;
   1:  PR[91,1] = PR[90,1] + -38.124;
   1:  PR[91,2] = PR[90,2] + -12.286;
   1:L PR[91] R[100]mm/sec CNT100;
   1:  PR[91,1] = PR[90,1] + -35.177;
   1:  PR[91,2] = PR[90,2] + -15.250;
   1:L PR[91] R[100]mm/sec CNT100;
   1:  PR[91,1] = PR[90,1] + -31.637;
   1:  PR[91,2] = PR[90,2] + -17.501;
   1:L PR[91] R[100]mm/sec CNT100;
   1:  PR[91,1] = PR[90,1] + -29.583;
   1:  PR[91,2] = PR[90,2] + -18.228;
   1:L PR[91] R[100]mm/sec CNT100;
   1:  PR[91,1] = PR[90,1] + -27.663;
   1:  PR[91,2] = PR[90,2] + -18.928;
   1:L PR[91] R[100]mm/sec CNT100;
   1:  PR[91,1] = PR[90,1] + -25.725;
   1:  PR[91,2] = PR[90,2] + -19.160;
   1:L PR[91] R[100]mm/sec CNT100;
   1:  PR[91,1] = PR[90,1] + -23.460;
   1:  PR[91,2] = PR[90,2] + -19.455;
   1:L PR[91] R[100]mm/sec CNT100;
   1:  PR[91,1] = PR[90,1] + -21.772;
   1:  PR[91,2] = PR[90,2] + -19.279;
   1:L PR[91] R[100]mm/sec CNT100;
   1:  PR[91,1] = PR[90,1] + -19.230;
   1:  PR[91,2] = PR[90,2] + -19.043;
   1:L PR[91] R[100]mm/sec CNT100;
   1:  PR[91,1] = PR[90,1] + -17.879;
   1:  PR[91,2] = PR[90,2] + -18.587;
   1:L PR[91] R[100]mm/sec CNT100;
   1:  PR[91,1] = PR[90,1] + -15.178;
   1:  PR[91,2] = PR[90,2] + -17.708;
   1:L PR[91] R[100]mm/sec CNT100;
   1:  PR[91,1] = PR[90,1] + -11.528;
   1:  PR[91,2] = PR[90,2] + -15.508;
   1:L PR[91] R[100]mm/sec CNT100;
   1:  PR[91,1] = PR[90,1] + -8.458;
   1:  PR[91,2] = PR[90,2] + -12.546;
   1:L PR[91] R[100]mm/sec CNT100;
   1:  PR[91,1] = PR[90,1] + -6.135;
   1:  PR[91,2] = PR[90,2] + -8.970;
   1:L PR[91] R[100]mm/sec CNT100;
   1:  PR[91,1] = PR[90,1] + -4.693;
   1:  PR[91,2] = PR[90,2] + -4.972;
   1:L PR[91] R[100]mm/sec CNT100;
   1:  PR[91,1] = PR[90,1] + -4.248;
   1:  PR[91,2] = PR[90,2] + -0.740;
   1:L PR[91] R[100]mm/sec CNT100;
   1:  PR[91,1] = PR[90,1] + -4.260;
   1:  PR[91,2] = PR[90,2] + -0.638;
   1:L PR[91] R[100]mm/sec CNT100;
   1:  PR[91,1] = PR[90,1] + -4.247;
   1:  PR[91,2] = PR[90,2] + -0.309;
   1:L PR[91] R[100]mm/sec CNT100;
   1:  PR[91,1] = PR[90,1] + -4.689;
   1:  PR[91,2] = PR[90,2] + 3.503;
   1:L PR[91] R[100]mm/sec CNT100;
   1:  PR[91,1] = PR[90,1] + -6.135;
   1:  PR[91,2] = PR[90,2] + 7.511;
   1:L PR[91] R[100]mm/sec CNT100;
   1:  PR[91,1] = PR[90,1] + -8.458;
   1:  PR[91,2] = PR[90,2] + 11.087;
   1:L PR[91] R[100]mm/sec CNT100;
   1:  PR[91,1] = PR[90,1] + -11.533;
   1:  PR[91,2] = PR[90,2] + 14.054;
   1:L PR[91] R[100]mm/sec CNT100;
   1:  PR[91,1] = PR[90,1] + -12.346;
   1:  PR[91,2] = PR[90,2] + 14.551;
   1:L PR[91] R[100]mm/sec CNT100TB   .50sec,CALL END_PUD;
   1:  PR[92] = PR[91];
   1:  PR[92,3] = PR[92,3] + 20;
   1:J PR[92] 10% FINE;
   1:  PR[91,1] = PR[90,1] + -53.021;
   1:  PR[91,2] = PR[90,2] + -4.699;
   1:  PR[92] = PR[91];
   1:  PR[92,3] = PR[92,3] + 20;
   1:J PR[92] 10% FINE;
   1:L PR[91] R[100]mm/sec CNT100;
   1:  CALL LASER_DRAHT_START;
   1:  PR[91,1] = PR[90,1] + -52.877;
   1:  PR[91,2] = PR[90,2] + -3.452;
   1:L PR[91] R[100]mm/sec CNT100;
   1:  PR[91,1] = PR[90,1] + -52.683;
   1:  PR[91,2] = PR[90,2] + -0.769;
   1:L PR[91] R[100]mm/sec CNT100;
   1:  PR[91,1] = PR[90,1] + -53.132;
   1:  PR[91,2] = PR[90,2] + 3.242;
   1:L PR[91] R[100]mm/sec CNT100;
   1:  PR[91,1] = PR[90,1] + -54.462;
   1:  PR[91,2] = PR[90,2] + 7.021;
   1:L PR[91] R[100]mm/sec CNT100;
   1:  PR[91,1] = PR[90,1] + -56.604;
   1:  PR[91,2] = PR[90,2] + 10.437;
   1:L PR[91] R[100]mm/sec CNT100;
   1:  PR[91,1] = PR[90,1] + -59.447;
   1:  PR[91,2] = PR[90,2] + 13.338;
   1:L PR[91] R[100]mm/sec CNT100;
   1:  PR[91,1] = PR[90,1] + -60.836;
   1:  PR[91,2] = PR[90,2] + 14.269;
   1:L PR[91] R[100]mm/sec CNT100;
   1:  PR[91,1] = PR[90,1] + -62.844;
   1:  PR[91,2] = PR[90,2] + 15.588;
   1:L PR[91] R[100]mm/sec CNT100;
   1:  PR[91,1] = PR[90,1] + -65.077;
   1:  PR[91,2] = PR[90,2] + 16.491;
   1:L PR[91] R[100]mm/sec CNT100;
   1:  PR[91,1] = PR[90,1] + -66.638;
   1:  PR[91,2] = PR[90,2] + 17.105;
   1:L PR[91] R[100]mm/sec CNT100;
   1:  PR[91,1] = PR[90,1] + -70.671;
   1:  PR[91,2] = PR[90,2] + 17.834;
   1:L PR[91] R[100]mm/sec CNT100;
   1:  PR[91,1] = PR[90,1] + -74.749;
   1:  PR[91,2] = PR[90,2] + 17.750;
   1:L PR[91] R[100]mm/sec CNT100;
   1:  PR[91,1] = PR[90,1] + -78.684;
   1:  PR[91,2] = PR[90,2] + 16.871;
   1:L PR[91] R[100]mm/sec CNT100;
   1:  PR[91,1] = PR[90,1] + -82.248;
   1:  PR[91,2] = PR[90,2] + 15.256;
   1:L PR[91] R[100]mm/sec CNT100;
   1:  PR[91,1] = PR[90,1] + -85.392;
   1:  PR[91,2] = PR[90,2] + 12.958;
   1:L PR[91] R[100]mm/sec CNT100;
   1:  PR[91,1] = PR[90,1] + -87.981;
   1:  PR[91,2] = PR[90,2] + 10.077;
   1:L PR[91] R[100]mm/sec CNT100;
   1:  PR[91,1] = PR[90,1] + -89.911;
   1:  PR[91,2] = PR[90,2] + 6.739;
   1:L PR[91] R[100]mm/sec CNT100;
   1:  PR[91,1] = PR[90,1] + -91.101;
   1:  PR[91,2] = PR[90,2] + 3.084;
   1:L PR[91] R[100]mm/sec CNT100;
   1:  PR[91,1] = PR[90,1] + -91.213;
   1:  PR[91,2] = PR[90,2] + 2.037;
   1:L PR[91] R[100]mm/sec CNT100;
   1:  PR[91,1] = PR[90,1] + -91.473;
   1:  PR[91,2] = PR[90,2] + 0.383;
   1:L PR[91] R[100]mm/sec CNT100;
   1:  PR[91,1] = PR[90,1] + -91.586;
   1:  PR[91,2] = PR[90,2] + -0.678;
   1:L PR[91] R[100]mm/sec CNT100;
   1:  PR[91,1] = PR[90,1] + -91.419;
   1:  PR[91,2] = PR[90,2] + -1.736;
   1:L PR[91] R[100]mm/sec CNT100;
   1:  PR[91,1] = PR[90,1] + -91.277;
   1:  PR[91,2] = PR[90,2] + -2.342;
   1:L PR[91] R[100]mm/sec CNT100;
   1:  PR[91,1] = PR[90,1] + -91.046;
   1:  PR[91,2] = PR[90,2] + -4.545;
   1:L PR[91] R[100]mm/sec CNT100;
   1:  PR[91,1] = PR[90,1] + -90.520;
   1:  PR[91,2] = PR[90,2] + -6.151;
   1:L PR[91] R[100]mm/sec CNT100;
   1:  PR[91,1] = PR[90,1] + -89.854;
   1:  PR[91,2] = PR[90,2] + -8.202;
   1:L PR[91] R[100]mm/sec CNT100;
   1:  PR[91,1] = PR[90,1] + -87.918;
   1:  PR[91,2] = PR[90,2] + -11.542;
   1:L PR[91] R[100]mm/sec CNT100;
   1:  PR[91,1] = PR[90,1] + -85.320;
   1:  PR[91,2] = PR[90,2] + -14.427;
   1:L PR[91] R[100]mm/sec CNT100;
   1:  PR[91,1] = PR[90,1] + -82.165;
   1:  PR[91,2] = PR[90,2] + -16.729;
   1:L PR[91] R[100]mm/sec CNT100;
   1:  PR[91,1] = PR[90,1] + -78.585;
   1:  PR[91,2] = PR[90,2] + -18.350;
   1:L PR[91] R[100]mm/sec CNT100;
   1:  PR[91,1] = PR[90,1] + -74.729;
   1:  PR[91,2] = PR[90,2] + -19.214;
   1:L PR[91] R[100]mm/sec CNT100;
   1:  PR[91,1] = PR[90,1] + -70.750;
   1:  PR[91,2] = PR[90,2] + -19.278;
   1:L PR[91] R[100]mm/sec CNT100;
   1:  PR[91,1] = PR[90,1] + -66.695;
   1:  PR[91,2] = PR[90,2] + -18.552;
   1:L PR[91] R[100]mm/sec CNT100;
   1:  PR[91,1] = PR[90,1] + -63.514;
   1:  PR[91,2] = PR[90,2] + -17.287;
   1:L PR[91] R[100]mm/sec CNT100;
   1:  PR[91,1] = PR[90,1] + -62.844;
   1:  PR[91,2] = PR[90,2] + -17.032;
   1:L PR[91] R[100]mm/sec CNT100;
   1:  PR[91,1] = PR[90,1] + -60.434;
   1:  PR[91,2] = PR[90,2] + -15.440;
   1:L PR[91] R[100]mm/sec CNT100;
   1:  PR[91,1] = PR[90,1] + -59.408;
   1:  PR[91,2] = PR[90,2] + -14.784;
   1:L PR[91] R[100]mm/sec CNT100;
   1:  PR[91,1] = PR[90,1] + -57.744;
   1:  PR[91,2] = PR[90,2] + -13.089;
   1:L PR[91] R[100]mm/sec CNT100;
   1:  PR[91,1] = PR[90,1] + -56.537;
   1:  PR[91,2] = PR[90,2] + -11.891;
   1:L PR[91] R[100]mm/sec CNT100;
   1:  PR[91,1] = PR[90,1] + -55.519;
   1:  PR[91,2] = PR[90,2] + -10.270;
   1:L PR[91] R[100]mm/sec CNT100;
   1:  PR[91,1] = PR[90,1] + -54.367;
   1:  PR[91,2] = PR[90,2] + -8.475;
   1:L PR[91] R[100]mm/sec CNT100;
   1:  PR[91,1] = PR[90,1] + -53.021;
   1:  PR[91,2] = PR[90,2] + -4.699;
   1:L PR[91] R[100]mm/sec CNT100TB   .50sec,CALL END_PUD;
   1:  PR[92] = PR[91];
   1:  PR[92,3] = PR[92,3] + 20;
   1:J PR[92] 10% FINE;
   1:  PR[91] = PR[90];
   1:  PR[91,1] = PR[90,1] + 87.268;
   1:  PR[91,2] = PR[90,2] + -12.439;
   1:  PR[91,3] = PR[90,3] + 28.795;
   1:  PR[92] = PR[91];
   1:  PR[92,3] = PR[92,3] + 20;
   1:J PR[92] 10% FINE;
   1:L PR[91] R[100]mm/sec CNT100;
   1:  CALL LASER_DRAHT_START;
   1:  PR[91,1] = PR[90,1] + 89.501;
   1:  PR[91,2] = PR[90,2] + -8.857;
   1:L PR[91] R[100]mm/sec CNT100;
   1:  PR[91,1] = PR[90,1] + 90.883;
   1:  PR[91,2] = PR[90,2] + -4.888;
   1:L PR[91] R[100]mm/sec CNT100;
   1:  PR[91,1] = PR[90,1] + 90.967;
   1:  PR[91,2] = PR[90,2] + -4.156;
   1:L PR[91] R[100]mm/sec CNT100;
   1:  PR[91,1] = PR[90,1] + 91.206;
   1:  PR[91,2] = PR[90,2] + -2.585;
   1:L PR[91] R[100]mm/sec CNT100;
   1:  PR[91,1] = PR[90,1] + 91.407;
   1:  PR[91,2] = PR[90,2] + -0.801;
   1:L PR[91] R[100]mm/sec CNT100;
   1:  PR[91,1] = PR[90,1] + 91.267;
   1:  PR[91,2] = PR[90,2] + -0.043;
   1:L PR[91] R[100]mm/sec CNT100;
   1:  PR[91,1] = PR[90,1] + 90.881;
   1:  PR[91,2] = PR[90,2] + 3.433;
   1:L PR[91] R[100]mm/sec CNT100;
   1:  PR[91,1] = PR[90,1] + 89.501;
   1:  PR[91,2] = PR[90,2] + 7.398;
   1:L PR[91] R[100]mm/sec CNT100;
   1:  PR[91,1] = PR[90,1] + 87.268;
   1:  PR[91,2] = PR[90,2] + 10.980;
   1:L PR[91] R[100]mm/sec CNT100;
   1:  PR[91,1] = PR[90,1] + 84.286;
   1:  PR[91,2] = PR[90,2] + 14.005;
   1:L PR[91] R[100]mm/sec CNT100;
   1:  PR[91,1] = PR[90,1] + 80.640;
   1:  PR[91,2] = PR[90,2] + 16.343;
   1:L PR[91] R[100]mm/sec CNT100;
   1:  PR[91,1] = PR[90,1] + 76.908;
   1:  PR[91,2] = PR[90,2] + 17.710;
   1:L PR[91] R[100]mm/sec CNT100;
   1:  PR[91,1] = PR[90,1] + 76.441;
   1:  PR[91,2] = PR[90,2] + 17.891;
   1:L PR[91] R[100]mm/sec CNT100;
   1:  PR[91,1] = PR[90,1] + 73.048;
   1:  PR[91,2] = PR[90,2] + 18.366;
   1:L PR[91] R[100]mm/sec CNT100;
   1:  PR[91,1] = PR[90,1] + 71.961;
   1:  PR[91,2] = PR[90,2] + 18.540;
   1:L PR[91] R[100]mm/sec CNT100;
   1:  PR[91,1] = PR[90,1] + 69.180;
   1:  PR[91,2] = PR[90,2] + 18.333;
   1:L PR[91] R[100]mm/sec CNT100;
   1:  PR[91,1] = PR[90,1] + 67.396;
   1:  PR[91,2] = PR[90,2] + 18.240;
   1:L PR[91] R[100]mm/sec CNT100;
   1:  PR[91,1] = PR[90,1] + 65.418;
   1:  PR[91,2] = PR[90,2] + 17.653;
   1:L PR[91] R[100]mm/sec CNT100;
   1:  PR[91,1] = PR[90,1] + 62.965;
   1:  PR[91,2] = PR[90,2] + 16.985;
   1:L PR[91] R[100]mm/sec CNT100;
   1:  PR[91,1] = PR[90,1] + 61.856;
   1:  PR[91,2] = PR[90,2] + 16.368;
   1:L PR[91] R[100]mm/sec CNT100;
   1:  PR[91,1] = PR[90,1] + 58.893;
   1:  PR[91,2] = PR[90,2] + 14.805;
   1:L PR[91] R[100]mm/sec CNT100;
   1:  PR[91,1] = PR[90,1] + 58.565;
   1:  PR[91,2] = PR[90,2] + 14.510;
   1:L PR[91] R[100]mm/sec CNT100;
   1:  PR[91,1] = PR[90,1] + 55.784;
   1:  PR[91,2] = PR[90,2] + 12.108;
   1:L PR[91] R[100]mm/sec CNT100;
   1:  PR[91,1] = PR[90,1] + 55.300;
   1:  PR[91,2] = PR[90,2] + 11.720;
   1:L PR[91] R[100]mm/sec CNT100;
   1:  PR[91,1] = PR[90,1] + 52.540;
   1:  PR[91,2] = PR[90,2] + 8.136;
   1:L PR[91] R[100]mm/sec CNT100;
   1:  PR[91,1] = PR[90,1] + 52.071;
   1:  PR[91,2] = PR[90,2] + 7.140;
   1:L PR[91] R[100]mm/sec CNT100;
   1:  PR[91,1] = PR[90,1] + 50.705;
   1:  PR[91,2] = PR[90,2] + 3.916;
   1:L PR[91] R[100]mm/sec CNT100;
   1:  PR[91,1] = PR[90,1] + 50.446;
   1:  PR[91,2] = PR[90,2] + 2.223;
   1:L PR[91] R[100]mm/sec CNT100;
   1:  PR[91,1] = PR[90,1] + 50.038;
   1:  PR[91,2] = PR[90,2] + -0.729;
   1:L PR[91] R[100]mm/sec CNT100;
   1:  PR[91,1] = PR[90,1] + 50.446;
   1:  PR[91,2] = PR[90,2] + -3.684;
   1:L PR[91] R[100]mm/sec CNT100;
   1:  PR[91,1] = PR[90,1] + 50.704;
   1:  PR[91,2] = PR[90,2] + -5.374;
   1:L PR[91] R[100]mm/sec CNT100;
